            'The trust relationship between this workstation and the primary domain failed.';
    Win32ErrorCodes.ERROR_TRUST_FAILURE:
        Win32ErrorCodeDescription := 'The network logon failed.';
    Win32ErrorCodes.RPC_S_CALL_IN_PROGRESS:
        Win32ErrorCodeDescription :=
            'A remote procedure call is already in progress for this thread.';
    Win32ErrorCodes.ERROR_NETLOGON_NOT_STARTED:
        Win32ErrorCodeDescription :=
            'An attempt was made to logon, but the network logon service was not started.';
    Win32ErrorCodes.ERROR_ACCOUNT_EXPIRED:
        Win32ErrorCodeDescription := 'The users account has expired.';
    Win32ErrorCodes.ERROR_REDIRECTOR_HAS_OPEN_HANDLES:
        Win32ErrorCodeDescription := 'The redirector is in use and cannot be unloaded.';
    Win32ErrorCodes.ERROR_PRINTER_DRIVER_ALREADY_INSTALLED:
        Win32ErrorCodeDescription := 'The specified printer driver is already installed.';
    Win32ErrorCodes.ERROR_UNKNOWN_PORT:
        Win32ErrorCodeDescription := 'The specified port is unknown.';
    Win32ErrorCodes.ERROR_UNKNOWN_PRINTER_DRIVER:
        Win32ErrorCodeDescription := 'The printer driver is unknown.';
    Win32ErrorCodes.ERROR_UNKNOWN_PRINTPROCESSOR:
        Win32ErrorCodeDescription := 'The print processor is unknown.';
    Win32ErrorCodes.ERROR_INVALID_SEPARATOR_FILE:
        Win32ErrorCodeDescription := 'The specified separator file is invalid.';
    Win32ErrorCodes.ERROR_INVALID_PRIORITY:
        Win32ErrorCodeDescription := 'The specified priority is invalid.';
    Win32ErrorCodes.ERROR_INVALID_PRINTER_NAME:
        Win32ErrorCodeDescription := 'The printer name is invalid.';
    Win32ErrorCodes.ERROR_PRINTER_ALREADY_EXISTS:
        Win32ErrorCodeDescription := 'The printer already exists.';
    Win32ErrorCodes.ERROR_INVALID_PRINTER_COMMAND:
        Win32ErrorCodeDescription := 'The printer command is invalid.';
    Win32ErrorCodes.ERROR_INVALID_DATATYPE:
        Win32ErrorCodeDescription := 'The specified datatype is invalid.';
    Win32ErrorCodes.ERROR_INVALID_ENVIRONMENT:
        Win32ErrorCodeDescription := 'The environment specified is invalid.';
    Win32ErrorCodes.RPC_S_NO_MORE_BINDINGS:
        Win32ErrorCodeDescription := 'There are no more bindings.';
    Win32ErrorCodes.ERROR_NOLOGON_INTERDOMAIN_TRUST_ACCOUNT:
        Win32ErrorCodeDescription := 'The account used is an interdomain trust account. Use your global user account or local user account to access this server.';
    Win32ErrorCodes.ERROR_NOLOGON_WORKSTATION_TRUST_ACCOUNT:
        Win32ErrorCodeDescription := 'The account used is a computer account. Use your global user account or local user account to access this server.';
    Win32ErrorCodes.ERROR_NOLOGON_SERVER_TRUST_ACCOUNT:
        Win32ErrorCodeDescription := 'The account used is a server trust account. Use your global user account or local user account to access this server.';
    Win32ErrorCodes.ERROR_DOMAIN_TRUST_INCONSISTENT:
        Win32ErrorCodeDescription := 'The name or security ID (SID) of the domain specified is inconsistent with the trust information for that domain.';
    Win32ErrorCodes.ERROR_SERVER_HAS_OPEN_HANDLES:
        Win32ErrorCodeDescription := 'The server is in use and cannot be unloaded.';
    Win32ErrorCodes.ERROR_RESOURCE_DATA_NOT_FOUND:
        Win32ErrorCodeDescription :=
            'The specified image file did not contain a resource section.';
    Win32ErrorCodes.ERROR_RESOURCE_TYPE_NOT_FOUND:
        Win32ErrorCodeDescription :=
            'The specified resource type cannot be found in the image file.';
    Win32ErrorCodes.ERROR_RESOURCE_NAME_NOT_FOUND:
        Win32ErrorCodeDescription :=
            'The specified resource name cannot be found in the image file.';
    Win32ErrorCodes.ERROR_RESOURCE_LANG_NOT_FOUND:
        Win32ErrorCodeDescription :=
            'The specified resource language ID cannot be found in the image file.';
    Win32ErrorCodes.ERROR_NOT_ENOUGH_QUOTA:
        Win32ErrorCodeDescription := 'Not enough quota is available to process this command.';
    Win32ErrorCodes.RPC_S_NO_INTERFACES:
        Win32ErrorCodeDescription := 'No interfaces have been registered.';
    Win32ErrorCodes.RPC_S_CALL_CANCELLED:
        Win32ErrorCodeDescription := 'The remote procedure call was cancelled.';
    Win32ErrorCodes.RPC_S_BINDING_INCOMPLETE:
        Win32ErrorCodeDescription :=
            'The binding handle does not contain all required information.';
    Win32ErrorCodes.RPC_S_COMM_FAILURE:
        Win32ErrorCodeDescription :=
            'A communications failure occurred during a remote procedure call.';
    Win32ErrorCodes.RPC_S_UNSUPPORTED_AUTHN_LEVEL:
        Win32ErrorCodeDescription := 'The requested authentication level is not supported.';
    Win32ErrorCodes.RPC_S_NO_PRINC_NAME:
        Win32ErrorCodeDescription := 'No principal name registered.';
    Win32ErrorCodes.RPC_S_NOT_RPC_ERROR:
        Win32ErrorCodeDescription := 'The error specified is not a valid Windows RPC error code.';
    Win32ErrorCodes.RPC_S_UUID_LOCAL_ONLY:
        Win32ErrorCodeDescription :=
            'A UUID that is valid only on this computer has been allocated.';
    Win32ErrorCodes.RPC_S_SEC_PKG_ERROR:
        Win32ErrorCodeDescription := 'A security package specific error occurred.';
    Win32ErrorCodes.RPC_S_NOT_CANCELLED:
        Win32ErrorCodeDescription := 'Thread is not canceled.';
    Win32ErrorCodes.RPC_X_INVALID_ES_ACTION:
        Win32ErrorCodeDescription := 'Invalid operation on the encoding/decoding handle.';
    Win32ErrorCodes.RPC_X_WRONG_ES_VERSION:
        Win32ErrorCodeDescription := 'Incompatible version of the serializing package.';
    Win32ErrorCodes.RPC_X_WRONG_STUB_VERSION:
        Win32ErrorCodeDescription := 'Incompatible version of the RPC stub.';
    Win32ErrorCodes.RPC_X_INVALID_PIPE_OBJECT:
        Win32ErrorCodeDescription := 'The RPC pipe object is invalid or corrupted.';
    Win32ErrorCodes.RPC_X_WRONG_PIPE_ORDER:
        Win32ErrorCodeDescription := 'An invalid operation was attempted on an RPC pipe object.';
    Win32ErrorCodes.RPC_X_WRONG_PIPE_VERSION:
        Win32ErrorCodeDescription := 'Unsupported RPC pipe version.';
    Win32ErrorCodes.RPC_S_GROUP_MEMBER_NOT_FOUND:
        Win32ErrorCodeDescription := 'The group member was not found.';
    Win32ErrorCodes.EPT_S_CANT_CREATE:
        Win32ErrorCodeDescription := 'The endpoint mapper database entry could not be created.';
    Win32ErrorCodes.RPC_S_INVALID_OBJECT:
        Win32ErrorCodeDescription :=
            'The object universal unique identifier (UUID) is the nil UUID.';
    Win32ErrorCodes.ERROR_INVALID_TIME:
        Win32ErrorCodeDescription := 'The specified time is invalid.';
    Win32ErrorCodes.ERROR_INVALID_FORM_NAME:
        Win32ErrorCodeDescription := 'The specified form name is invalid.';
    Win32ErrorCodes.ERROR_INVALID_FORM_SIZE:
        Win32ErrorCodeDescription := 'The specified form size is invalid.';
    Win32ErrorCodes.ERROR_ALREADY_WAITING:
        Win32ErrorCodeDescription := 'The specified printer handle is already being waited on';
    Win32ErrorCodes.ERROR_PRINTER_DELETED:
        Win32ErrorCodeDescription := 'The specified printer has been deleted.';
    Win32ErrorCodes.ERROR_INVALID_PRINTER_STATE:
        Win32ErrorCodeDescription := 'The state of the printer is invalid.';
    Win32ErrorCodes.ERROR_PASSWORD_MUST_CHANGE:
        Win32ErrorCodeDescription :=
            'The users password must be changed before logging on the first time.';
    Win32ErrorCodes.ERROR_DOMAIN_CONTROLLER_NOT_FOUND:
        Win32ErrorCodeDescription := 'Could not find the domain controller for this domain.';
    Win32ErrorCodes.ERROR_ACCOUNT_LOCKED_OUT:
        Win32ErrorCodeDescription :=
            'The referenced account is currently locked out and may not be logged on to.';
    Win32ErrorCodes.OR_INVALID_OXID:
        Win32ErrorCodeDescription := 'The object exporter specified was not found.';
    Win32ErrorCodes.OR_INVALID_OID:
        Win32ErrorCodeDescription := 'The object specified was not found.';
    Win32ErrorCodes.OR_INVALID_SET:
        Win32ErrorCodeDescription := 'The object resolver set specified was not found.';
    Win32ErrorCodes.RPC_S_SEND_INCOMPLETE:
        Win32ErrorCodeDescription := 'Some data remains to be sent in the request buffer.';
    Win32ErrorCodes.RPC_S_INVALID_ASYNC_HANDLE:
        Win32ErrorCodeDescription := 'Invalid asynchronous remote procedure call handle.';
    Win32ErrorCodes.RPC_S_INVALID_ASYNC_CALL:
        Win32ErrorCodeDescription := 'Invalid asynchronous RPC call handle for this operation.';
    Win32ErrorCodes.RPC_X_PIPE_CLOSED:
        Win32ErrorCodeDescription := 'The RPC pipe object has already been closed.';
    Win32ErrorCodes.RPC_X_PIPE_DISCIPLINE_ERROR:
        Win32ErrorCodeDescription := 'The RPC call completed before all pipes were processed.';
    Win32ErrorCodes.RPC_X_PIPE_EMPTY:
        Win32ErrorCodeDescription := 'No more data is available from the RPC pipe.';
    Win32ErrorCodes.ERROR_NO_SITENAME:
        Win32ErrorCodeDescription := 'No site name is available for this machine.';
    Win32ErrorCodes.ERROR_CANT_ACCESS_FILE:
        Win32ErrorCodeDescription := 'The file can not be accessed by the system.';
    Win32ErrorCodes.ERROR_CANT_RESOLVE_FILENAME:
        Win32ErrorCodeDescription := 'The name of the file cannot be resolved by the system.';
    Win32ErrorCodes.RPC_S_ENTRY_TYPE_MISMATCH:
        Win32ErrorCodeDescription := 'The entry is not of the expected type.';
    Win32ErrorCodes.RPC_S_NOT_ALL_OBJS_EXPORTED:
        Win32ErrorCodeDescription :=
            'Not all object UUIDs could be exported to the specified entry.';
    Win32ErrorCodes.RPC_S_INTERFACE_NOT_EXPORTED:
        Win32ErrorCodeDescription := 'Interface could not be exported to the specified entry.';
    Win32ErrorCodes.RPC_S_PROFILE_NOT_ADDED:
        Win32ErrorCodeDescription := 'The specified profile entry could not be added.';
    Win32ErrorCodes.RPC_S_PRF_ELT_NOT_ADDED:
        Win32ErrorCodeDescription := 'The specified profile element could not be added.';
    Win32ErrorCodes.RPC_S_PRF_ELT_NOT_REMOVED:
        Win32ErrorCodeDescription := 'The specified profile element could not be removed.';
    Win32ErrorCodes.RPC_S_GRP_ELT_NOT_ADDED:
        Win32ErrorCodeDescription := 'The group element could not be added.';
    Win32ErrorCodes.RPC_S_GRP_ELT_NOT_REMOVED:
        Win32ErrorCodeDescription := 'The group element could not be removed.';
    Win32ErrorCodes.ERROR_KM_DRIVER_BLOCKED:
        Win32ErrorCodeDescription := 'The printer driver is not compatible with a policy enabled on your computer that blocks NT 4.0 drivers.';
    Win32ErrorCodes.ERROR_INVALID_PIXEL_FORMAT:
        Win32ErrorCodeDescription := 'The pixel format is invalid.';
    Win32ErrorCodes.ERROR_BAD_DRIVER:
        Win32ErrorCodeDescription := 'The specified driver is invalid.';
    Win32ErrorCodes.ERROR_INVALID_WINDOW_STYLE:
        Win32ErrorCodeDescription :=
            'The window style or class attribute is invalid for this operation.';
    Win32ErrorCodes.ERROR_METAFILE_NOT_SUPPORTED:
        Win32ErrorCodeDescription := 'The requested metafile operation is not supported.';
    Win32ErrorCodes.ERROR_TRANSFORM_NOT_SUPPORTED:
        Win32ErrorCodeDescription := 'The requested transformation operation is not supported.';
    Win32ErrorCodes.ERROR_CLIPPING_NOT_SUPPORTED:
        Win32ErrorCodeDescription := 'The requested clipping operation is not supported.';
    Win32ErrorCodes.ERROR_INVALID_CMM:
        Win32ErrorCodeDescription := 'The specified color management module is invalid.';
    Win32ErrorCodes.ERROR_INVALID_PROFILE:
        Win32ErrorCodeDescription := 'The specified color profile is invalid.';
    Win32ErrorCodes.ERROR_TAG_NOT_FOUND:
        Win32ErrorCodeDescription := 'The specified tag was not found.';
    Win32ErrorCodes.ERROR_TAG_NOT_PRESENT:
        Win32ErrorCodeDescription := 'A required tag is not present.';
    Win32ErrorCodes.ERROR_DUPLICATE_TAG:
        Win32ErrorCodeDescription := 'The specified tag is already present.';
    Win32ErrorCodes.ERROR_PROFILE_NOT_ASSOCIATED_WITH_DEVICE:
        Win32ErrorCodeDescription :=
            'The specified color profile is not associated with any device.';
    Win32ErrorCodes.ERROR_PROFILE_NOT_FOUND:
        Win32ErrorCodeDescription := 'The specified color profile was not found.';
    Win32ErrorCodes.ERROR_INVALID_COLORSPACE:
        Win32ErrorCodeDescription := 'The specified color space is invalid.';
    Win32ErrorCodes.ERROR_ICM_NOT_ENABLED:
        Win32ErrorCodeDescription := 'Image Color Management is not enabled.';
    Win32ErrorCodes.ERROR_DELETING_ICM_XFORM:
        Win32ErrorCodeDescription := 'There was an error while deleting the color transform.';
    Win32ErrorCodes.ERROR_INVALID_TRANSFORM:
        Win32ErrorCodeDescription := 'The specified color transform is invalid.';
    Win32ErrorCodes.ERROR_COLORSPACE_MISMATCH:
        Win32ErrorCodeDescription :=
            'The specified transform does not match the bitmaps color space.';
    Win32ErrorCodes.ERROR_INVALID_COLORINDEX:
        Win32ErrorCodeDescription :=
            'The specified named color index is not present in the profile.';
    Win32ErrorCodes.ERROR_CONNECTED_OTHER_PASSWORD:
        Win32ErrorCodeDescription := 'The network connection was made successfully, but the user had to be prompted for a password other than the one originally specified.';
    Win32ErrorCodes.ERROR_BAD_USERNAME:
        Win32ErrorCodeDescription := 'The specified username is invalid.';
    Win32ErrorCodes.ERROR_NOT_CONNECTED:
        Win32ErrorCodeDescription := 'This network connection does not exist.';
    Win32ErrorCodes.ERROR_OPEN_FILES:
        Win32ErrorCodeDescription := 'This network connection has files open or requests pending.';
    Win32ErrorCodes.ERROR_ACTIVE_CONNECTIONS:
        Win32ErrorCodeDescription := 'Active connections still exist.';
    Win32ErrorCodes.ERROR_DEVICE_IN_USE:
        Win32ErrorCodeDescription :=
            'The device is in use by an active process and cannot be disconnected.';
    Win32ErrorCodes.ERROR_PKINIT_FAILURE:
        Win32ErrorCodeDescription := 'The kerberos protocol encountered an error while validating the KDC certificate during smartcard logon.';
    Win32ErrorCodes.ERROR_SMARTCARD_SUBSYSTEM_FAILURE:
        Win32ErrorCodeDescription := 'The kerberos protocol encountered an error while attempting to utilize the smartcard subsystem.';
    Win32ErrorCodes.ERROR_UNKNOWN_PRINT_MONITOR:
        Win32ErrorCodeDescription := 'The specified print monitor is unknown.';
    Win32ErrorCodes.ERROR_PRINTER_DRIVER_IN_USE:
        Win32ErrorCodeDescription := 'The specified printer driver is currently in use.';
    Win32ErrorCodes.ERROR_SPOOL_FILE_NOT_FOUND:
        Win32ErrorCodeDescription := 'The spool file was not found.';
    Win32ErrorCodes.ERROR_SPL_NO_STARTDOC:
        Win32ErrorCodeDescription := 'A StartDocPrinter call was not issued.';
    Win32ErrorCodes.ERROR_SPL_NO_ADDJOB:
        Win32ErrorCodeDescription := 'An AddJob call was not issued.';
    Win32ErrorCodes.ERROR_PRINT_PROCESSOR_ALREADY_INSTALLED:
        Win32ErrorCodeDescription := 'The specified print processor has already been installed.';
    Win32ErrorCodes.ERROR_PRINT_MONITOR_ALREADY_INSTALLED:
        Win32ErrorCodeDescription := 'The specified print monitor has already been installed.';
    Win32ErrorCodes.ERROR_INVALID_PRINT_MONITOR:
        Win32ErrorCodeDescription :=
            'The specified print monitor does not have the required functions.';
    Win32ErrorCodes.ERROR_PRINT_MONITOR_IN_USE:
        Win32ErrorCodeDescription := 'The specified print monitor is currently in use.';
    Win32ErrorCodes.ERROR_PRINTER_HAS_JOBS_QUEUED:
        Win32ErrorCodeDescription :=
            'The requested operation is not allowed when there are jobs queued to the printer.';
    Win32ErrorCodes.ERROR_SUCCESS_REBOOT_REQUIRED:
        Win32ErrorCodeDescription := 'The requested operation is successful. Changes will not be effective until the system is rebooted.';
    Win32ErrorCodes.ERROR_SUCCESS_RESTART_REQUIRED:
        Win32ErrorCodeDescription := 'The requested operation is successful. Changes will not be effective until the service is restarted.';
    Win32ErrorCodes.ERROR_PRINTER_NOT_FOUND:
        Win32ErrorCodeDescription := 'No printers were found.';
    Win32ErrorCodes.ERROR_WINS_INTERNAL:
        Win32ErrorCodeDescription := 'WINS encountered an error while processing the command.';
    Win32ErrorCodes.ERROR_CAN_NOT_DEL_LOCAL_WINS:
        Win32ErrorCodeDescription := 'The local WINS can not be deleted.';
    Win32ErrorCodes.ERROR_STATIC_INIT:
        Win32ErrorCodeDescription := 'The importation from the file failed.';
    Win32ErrorCodes.ERROR_INC_BACKUP:
        Win32ErrorCodeDescription := 'The backup failed. Was a full backup done before?';
    Win32ErrorCodes.ERROR_FULL_BACKUP:
        Win32ErrorCodeDescription :=
            'The backup failed. Check the directory to which you are backing the database.';
    Win32ErrorCodes.ERROR_REC_NON_EXISTENT:
        Win32ErrorCodeDescription := 'The name does not exist in the WINS database.';
    Win32ErrorCodes.ERROR_RPL_NOT_ALLOWED:
        Win32ErrorCodeDescription := 'Replication with a nonconfigured partner is not allowed.';
    Win32ErrorCodes.ERROR_DHCP_ADDRESS_CONFLICT:
        Win32ErrorCodeDescription := 'The DHCP client has obtained an IP address that is already in use on the network. The local interface will be disabled until the DHCP client can obtain a new address.';
    Win32ErrorCodes.ERROR_WMI_GUID_NOT_FOUND:
        Win32ErrorCodeDescription :=
            'The GUID passed was not recognized as valid by a WMI data provider.';
    Win32ErrorCodes.ERROR_WMI_INSTANCE_NOT_FOUND:
        Win32ErrorCodeDescription :=
            'The instance name passed was not recognized as valid by a WMI data provider.';
    Win32ErrorCodes.ERROR_WMI_ITEMID_NOT_FOUND:
        Win32ErrorCodeDescription :=
            'The data item ID passed was not recognized as valid by a WMI data provider.';
    Win32ErrorCodes.ERROR_WMI_TRY_AGAIN:
        Win32ErrorCodeDescription :=
            'The WMI request could not be completed and should be retried.';
    Win32ErrorCodes.ERROR_WMI_DP_NOT_FOUND:
        Win32ErrorCodeDescription := 'The WMI data provider could not be located.';
    Win32ErrorCodes.ERROR_WMI_UNRESOLVED_INSTANCE_REF:
        Win32ErrorCodeDescription :=
            'The WMI data provider references an instance set that has not been registered.';
    Win32ErrorCodes.ERROR_WMI_ALREADY_ENABLED:
        Win32ErrorCodeDescription :=
            'The WMI data block or event notification has already been enabled.';
    Win32ErrorCodes.ERROR_WMI_GUID_DISCONNECTED:
        Win32ErrorCodeDescription := 'The WMI data block is no longer available.';
    Win32ErrorCodes.ERROR_WMI_SERVER_UNAVAILABLE:
        Win32ErrorCodeDescription := 'The WMI data service is not available.';
    Win32ErrorCodes.ERROR_WMI_DP_FAILED:
        Win32ErrorCodeDescription := 'The WMI data provider failed to carry out the request.';
    Win32ErrorCodes.ERROR_WMI_INVALID_MOF:
        Win32ErrorCodeDescription := 'The WMI MOF information is not valid.';
    Win32ErrorCodes.ERROR_WMI_INVALID_REGINFO:
        Win32ErrorCodeDescription := 'The WMI registration information is not valid.';
    Win32ErrorCodes.ERROR_WMI_ALREADY_DISABLED:
        Win32ErrorCodeDescription :=
            'The WMI data block or event notification has already been disabled.';
    Win32ErrorCodes.ERROR_WMI_READ_ONLY:
        Win32ErrorCodeDescription := 'The WMI data item or data block is read only.';
    Win32ErrorCodes.ERROR_WMI_SET_FAILURE:
        Win32ErrorCodeDescription := 'The WMI data item or data block could not be changed.';
    Win32ErrorCodes.ERROR_INVALID_MEDIA:
        Win32ErrorCodeDescription := 'The media identifier does not represent a valid medium.';
    Win32ErrorCodes.ERROR_INVALID_LIBRARY:
        Win32ErrorCodeDescription := 'The library identifier does not represent a valid library.';
    Win32ErrorCodes.ERROR_INVALID_MEDIA_POOL:
        Win32ErrorCodeDescription :=
            'The media pool identifier does not represent a valid media pool.';
    Win32ErrorCodes.ERROR_DRIVE_MEDIA_MISMATCH:
        Win32ErrorCodeDescription :=
            'The drive and medium are not compatible or exist in different libraries.';
    Win32ErrorCodes.ERROR_MEDIA_OFFLINE:
        Win32ErrorCodeDescription := 'The medium currently exists in an offline library and must be online to perform this operation.';
    Win32ErrorCodes.ERROR_LIBRARY_OFFLINE:
        Win32ErrorCodeDescription := 'The operation cannot be performed on an offline library.';
    Win32ErrorCodes.ERROR_EMPTY:
        Win32ErrorCodeDescription := 'The library, drive, or media pool is empty.';
    Win32ErrorCodes.ERROR_NOT_EMPTY:
        Win32ErrorCodeDescription :=
            'The library, drive, or media pool must be empty to perform this operation.';
    Win32ErrorCodes.ERROR_MEDIA_UNAVAILABLE:
        Win32ErrorCodeDescription :=
            'No media is currently available in this media pool or library.';
    Win32ErrorCodes.ERROR_RESOURCE_DISABLED:
        Win32ErrorCodeDescription := 'A resource required for this operation is disabled.';
    Win32ErrorCodes.ERROR_INVALID_CLEANER:
        Win32ErrorCodeDescription := 'The media identifier does not represent a valid cleaner.';
    Win32ErrorCodes.ERROR_UNABLE_TO_CLEAN:
        Win32ErrorCodeDescription := 'The drive cannot be cleaned or does not support cleaning.';
    Win32ErrorCodes.ERROR_OBJECT_NOT_FOUND:
        Win32ErrorCodeDescription := 'The object identifier does not represent a valid object.';
    Win32ErrorCodes.ERROR_DATABASE_FAILURE:
        Win32ErrorCodeDescription := 'Unable to read from or write to the database.';
    Win32ErrorCodes.ERROR_DATABASE_FULL:
        Win32ErrorCodeDescription := 'The database is full.';
    Win32ErrorCodes.ERROR_MEDIA_INCOMPATIBLE:
        Win32ErrorCodeDescription := 'The medium is not compatible with the device or media pool.';
    Win32ErrorCodes.ERROR_RESOURCE_NOT_PRESENT:
        Win32ErrorCodeDescription := 'The resource required for this operation does not exist.';
    Win32ErrorCodes.ERROR_INVALID_OPERATION:
        Win32ErrorCodeDescription := 'The operation identifier is not valid.';
    Win32ErrorCodes.ERROR_MEDIA_NOT_AVAILABLE:
        Win32ErrorCodeDescription := 'The media is not mounted or ready for use.';
    Win32ErrorCodes.ERROR_DEVICE_NOT_AVAILABLE:
        Win32ErrorCodeDescription := 'The device is not ready for use.';
    Win32ErrorCodes.ERROR_REQUEST_REFUSED:
        Win32ErrorCodeDescription := 'The operator or administrator has refused the request.';
    Win32ErrorCodes.ERROR_INVALID_DRIVE_OBJECT:
        Win32ErrorCodeDescription := 'The drive identifier does not represent a valid drive.';
    Win32ErrorCodes.ERROR_LIBRARY_FULL:
        Win32ErrorCodeDescription := 'Library is full. No slot is available for use.';
    Win32ErrorCodes.ERROR_MEDIUM_NOT_ACCESSIBLE:
        Win32ErrorCodeDescription := 'The transport cannot access the medium.';
    Win32ErrorCodes.ERROR_UNABLE_TO_LOAD_MEDIUM:
        Win32ErrorCodeDescription := 'Unable to load the medium into the drive.';
    Win32ErrorCodes.ERROR_UNABLE_TO_INVENTORY_DRIVE:
        Win32ErrorCodeDescription := 'Unable to retrieve status about the drive.';
    Win32ErrorCodes.ERROR_UNABLE_TO_INVENTORY_SLOT:
        Win32ErrorCodeDescription := 'Unable to retrieve status about the slot.';
    Win32ErrorCodes.ERROR_UNABLE_TO_INVENTORY_TRANSPORT:
        Win32ErrorCodeDescription := 'Unable to retrieve status about the transport.';
    Win32ErrorCodes.ERROR_TRANSPORT_FULL:
        Win32ErrorCodeDescription := 'Cannot use the transport because it is already in use.';
    Win32ErrorCodes.ERROR_CONTROLLING_IEPORT:
        Win32ErrorCodeDescription := 'Unable to open or close the inject/eject port.';
    Win32ErrorCodes.ERROR_UNABLE_TO_EJECT_MOUNTED_MEDIA:
        Win32ErrorCodeDescription := 'Unable to eject the media because it is in a drive.';
    Win32ErrorCodes.ERROR_CLEANER_SLOT_SET:
        Win32ErrorCodeDescription := 'A cleaner slot is already reserved.';
    Win32ErrorCodes.ERROR_CLEANER_SLOT_NOT_SET:
        Win32ErrorCodeDescription := 'A cleaner slot is not reserved.';
    Win32ErrorCodes.ERROR_CLEANER_CARTRIDGE_SPENT:
        Win32ErrorCodeDescription :=
            'The cleaner cartridge has performed the maximum number of drive cleanings.';
    Win32ErrorCodes.ERROR_UNEXPECTED_OMID:
        Win32ErrorCodeDescription := 'Unexpected on-medium identifier.';
    Win32ErrorCodes.ERROR_CANT_DELETE_LAST_ITEM:
        Win32ErrorCodeDescription :=
            'The last remaining item in this group or resource cannot be deleted.';
    Win32ErrorCodes.ERROR_MESSAGE_EXCEEDS_MAX_SIZE:
        Win32ErrorCodeDescription :=
            'The message provided exceeds the maximum size allowed for this parameter.';
    Win32ErrorCodes.ERROR_VOLUME_CONTAINS_SYS_FILES:
        Win32ErrorCodeDescription := 'The volume contains system or paging files.';
    Win32ErrorCodes.ERROR_INDIGENOUS_TYPE:
        Win32ErrorCodeDescription := 'The media type cannot be removed from this library since at least one drive in the library reports it can support this media type.';
    Win32ErrorCodes.ERROR_NO_SUPPORTING_DRIVES:
        Win32ErrorCodeDescription := 'This offline media cannot be mounted on this system since no enabled drives are present which can be used.';
    Win32ErrorCodes.ERROR_CLEANER_CARTRIDGE_INSTALLED:
        Win32ErrorCodeDescription := 'A cleaner cartridge is present in the tape library.';
    Win32ErrorCodes.ERROR_FILE_OFFLINE:
        Win32ErrorCodeDescription := 'The remote storage service was not able to recall the file.';
    Win32ErrorCodes.ERROR_REMOTE_STORAGE_NOT_ACTIVE:
        Win32ErrorCodeDescription := 'The remote storage service is not operational at this time.';
    Win32ErrorCodes.ERROR_REMOTE_STORAGE_MEDIA_ERROR:
        Win32ErrorCodeDescription := 'The remote storage service encountered a media error.';
    Win32ErrorCodes.ERROR_NOT_A_REPARSE_POINT:
        Win32ErrorCodeDescription := 'The file or directory is not a reparse point.';
    Win32ErrorCodes.ERROR_REPARSE_ATTRIBUTE_CONFLICT:
        Win32ErrorCodeDescription := 'The reparse point attribute cannot be set because it conflicts with an existing attribute.';
    Win32ErrorCodes.ERROR_INVALID_REPARSE_DATA:
        Win32ErrorCodeDescription := 'The data present in the reparse point buffer is invalid.';
    Win32ErrorCodes.ERROR_REPARSE_TAG_INVALID:
        Win32ErrorCodeDescription := 'The tag present in the reparse point buffer is invalid.';
    Win32ErrorCodes.ERROR_REPARSE_TAG_MISMATCH:
        Win32ErrorCodeDescription := 'There is a mismatch between the tag specified in the request and the tag present in the reparse point.';
    Win32ErrorCodes.ERROR_VOLUME_NOT_SIS_ENABLED:
        Win32ErrorCodeDescription := 'Single Instance Storage is not available on this volume.';
    Win32ErrorCodes.ERROR_DEPENDENT_RESOURCE_EXISTS:
        Win32ErrorCodeDescription := 'The cluster resource cannot be moved to another group because other resources are dependent on it.';
    Win32ErrorCodes.ERROR_DEPENDENCY_NOT_FOUND:
        Win32ErrorCodeDescription := 'The cluster resource dependency cannot be found.';
    Win32ErrorCodes.ERROR_DEPENDENCY_ALREADY_EXISTS:
        Win32ErrorCodeDescription := 'The cluster resource cannot be made dependent on the specified resource because it is already dependent.';
    Win32ErrorCodes.ERROR_RESOURCE_NOT_ONLINE:
        Win32ErrorCodeDescription := 'The cluster resource is not online.';
    Win32ErrorCodes.ERROR_HOST_NODE_NOT_AVAILABLE:
        Win32ErrorCodeDescription := 'A cluster node is not available for this operation.';
    Win32ErrorCodes.ERROR_RESOURCE_NOT_AVAILABLE:
        Win32ErrorCodeDescription := 'The cluster resource is not available.';
    Win32ErrorCodes.ERROR_RESOURCE_NOT_FOUND:
        Win32ErrorCodeDescription := 'The cluster resource could not be found.';
    Win32ErrorCodes.ERROR_SHUTDOWN_CLUSTER:
        Win32ErrorCodeDescription := 'The cluster is being shut down.';
    Win32ErrorCodes.ERROR_CANT_EVICT_ACTIVE_NODE:
        Win32ErrorCodeDescription :=
            'A cluster node cannot be evicted from the cluster unless the node is down.';
    Win32ErrorCodes.ERROR_OBJECT_ALREADY_EXISTS:
        Win32ErrorCodeDescription := 'The object already exists.';
    Win32ErrorCodes.ERROR_OBJECT_IN_LIST:
        Win32ErrorCodeDescription := 'The object is already in the list.';
    Win32ErrorCodes.ERROR_GROUP_NOT_AVAILABLE:
        Win32ErrorCodeDescription := 'The cluster group is not available for any new requests.';
    Win32ErrorCodes.ERROR_GROUP_NOT_FOUND:
        Win32ErrorCodeDescription := 'The cluster group could not be found.';
    Win32ErrorCodes.ERROR_GROUP_NOT_ONLINE:
        Win32ErrorCodeDescription :=
            'The operation could not be completed because the cluster group is not online.';
    Win32ErrorCodes.ERROR_HOST_NODE_NOT_RESOURCE_OWNER:
        Win32ErrorCodeDescription := 'The cluster node is not the owner of the resource.';
    Win32ErrorCodes.ERROR_HOST_NODE_NOT_GROUP_OWNER:
        Win32ErrorCodeDescription := 'The cluster node is not the owner of the group.';
    Win32ErrorCodes.ERROR_RESMON_CREATE_FAILED:
        Win32ErrorCodeDescription :=
            'The cluster resource could not be created in the specified resource monitor.';
    Win32ErrorCodes.ERROR_RESMON_ONLINE_FAILED:
        Win32ErrorCodeDescription :=
            'The cluster resource could not be brought online by the resource monitor.';
    Win32ErrorCodes.ERROR_RESOURCE_ONLINE:
        Win32ErrorCodeDescription :=
            'The operation could not be completed because the cluster resource is online.';
    Win32ErrorCodes.ERROR_QUORUM_RESOURCE:
        Win32ErrorCodeDescription := 'The cluster resource could not be deleted or brought offline because it is the quorum resource.';
    Win32ErrorCodes.ERROR_NOT_QUORUM_CAPABLE:
        Win32ErrorCodeDescription := 'The cluster could not make the specified resource a quorum resource because it is not capable of being a quorum resource.';
    Win32ErrorCodes.ERROR_CLUSTER_SHUTTING_DOWN:
        Win32ErrorCodeDescription := 'The cluster software is shutting down.';
    Win32ErrorCodes.ERROR_INVALID_STATE:
        Win32ErrorCodeDescription :=
            'The group or resource is not in the correct state to perform the requested operation.';
    Win32ErrorCodes.ERROR_RESOURCE_PROPERTIES_STORED:
        Win32ErrorCodeDescription := 'The properties were stored but not all changes will take effect until the next time the resource is brought online.';
    Win32ErrorCodes.ERROR_NOT_QUORUM_CLASS:
        Win32ErrorCodeDescription := 'The cluster could not make the specified resource a quorum resource because it does not belong to a shared storage class.';
    Win32ErrorCodes.ERROR_CORE_RESOURCE:
        Win32ErrorCodeDescription :=
            'The cluster resource could not be deleted since it is a core resource.';
    Win32ErrorCodes.ERROR_QUORUM_RESOURCE_ONLINE_FAILED:
        Win32ErrorCodeDescription := 'The quorum resource failed to come online.';
    Win32ErrorCodes.ERROR_QUORUMLOG_OPEN_FAILED:
        Win32ErrorCodeDescription :=
            'The quorum log could not be created or mounted successfully.';
    Win32ErrorCodes.ERROR_CLUSTERLOG_CORRUPT:
        Win32ErrorCodeDescription := 'The cluster log is corrupt.';
    Win32ErrorCodes.ERROR_CLUSTERLOG_RECORD_EXCEEDS_MAXSIZE:
        Win32ErrorCodeDescription :=
            'The record could not be written to the cluster log since it exceeds the maximum size.';
    Win32ErrorCodes.ERROR_CLUSTERLOG_EXCEEDS_MAXSIZE:
        Win32ErrorCodeDescription := 'The cluster log exceeds its maximum size.';
    Win32ErrorCodes.ERROR_CLUSTERLOG_CHKPOINT_NOT_FOUND:
        Win32ErrorCodeDescription := 'No checkpoint record was found in the cluster log.';
    Win32ErrorCodes.ERROR_CLUSTERLOG_NOT_ENOUGH_SPACE:
        Win32ErrorCodeDescription :=
            'The minimum required disk space needed for logging is not available.';
    Win32ErrorCodes.ERROR_QUORUM_OWNER_ALIVE:
        Win32ErrorCodeDescription := 'The cluster node failed to take control of the quorum resource because the resource is owned by another active node.';
    Win32ErrorCodes.ERROR_NETWORK_NOT_AVAILABLE:
        Win32ErrorCodeDescription := 'A cluster network is not available for this operation.';
    Win32ErrorCodes.ERROR_NODE_NOT_AVAILABLE:
        Win32ErrorCodeDescription := 'A cluster node is not available for this operation.';
    Win32ErrorCodes.ERROR_ALL_NODES_NOT_AVAILABLE:
        Win32ErrorCodeDescription :=
            'All cluster nodes must be running to perform this operation.';
    Win32ErrorCodes.ERROR_RESOURCE_FAILED:
        Win32ErrorCodeDescription := 'A cluster resource failed.';
    Win32ErrorCodes.ERROR_CLUSTER_INVALID_NODE:
        Win32ErrorCodeDescription := 'The cluster node is not valid.';
    Win32ErrorCodes.ERROR_CLUSTER_NODE_EXISTS:
        Win32ErrorCodeDescription := 'The cluster node already exists.';
    Win32ErrorCodes.ERROR_CLUSTER_JOIN_IN_PROGRESS:
        Win32ErrorCodeDescription := 'A node is in the process of joining the cluster.';
    Win32ErrorCodes.ERROR_CLUSTER_NODE_NOT_FOUND:
        Win32ErrorCodeDescription := 'The cluster node was not found.';
    Win32ErrorCodes.ERROR_CLUSTER_LOCAL_NODE_NOT_FOUND:
        Win32ErrorCodeDescription := 'The cluster local node information was not found.';
    Win32ErrorCodes.ERROR_CLUSTER_NETWORK_EXISTS:
        Win32ErrorCodeDescription := 'The cluster network already exists.';
    Win32ErrorCodes.ERROR_CLUSTER_NETWORK_NOT_FOUND:
        Win32ErrorCodeDescription := 'The cluster network was not found.';
    Win32ErrorCodes.ERROR_CLUSTER_NETINTERFACE_EXISTS:
        Win32ErrorCodeDescription := 'The cluster network interface already exists.';
    Win32ErrorCodes.ERROR_CLUSTER_NETINTERFACE_NOT_FOUND:
        Win32ErrorCodeDescription := 'The cluster network interface was not found.';
    Win32ErrorCodes.ERROR_CLUSTER_INVALID_REQUEST:
        Win32ErrorCodeDescription := 'The cluster request is not valid for this object.';
    Win32ErrorCodes.ERROR_CLUSTER_INVALID_NETWORK_PROVIDER:
        Win32ErrorCodeDescription := 'The cluster network provider is not valid.';
    Win32ErrorCodes.ERROR_CLUSTER_NODE_DOWN:
        Win32ErrorCodeDescription := 'The cluster node is down.';
    Win32ErrorCodes.ERROR_CLUSTER_NODE_UNREACHABLE:
        Win32ErrorCodeDescription := 'The cluster node is not reachable.';
    Win32ErrorCodes.ERROR_CLUSTER_NODE_NOT_MEMBER:
        Win32ErrorCodeDescription := 'The cluster node is not a member of the cluster.';
    Win32ErrorCodes.ERROR_CLUSTER_JOIN_NOT_IN_PROGRESS:
        Win32ErrorCodeDescription := 'A cluster join operation is not in progress.';
    Win32ErrorCodes.ERROR_CLUSTER_INVALID_NETWORK:
        Win32ErrorCodeDescription := 'The cluster network is not valid.';
    Win32ErrorCodes.ERROR_CLUSTER_NODE_UP:
        Win32ErrorCodeDescription := 'The cluster node is up.';
    Win32ErrorCodes.ERROR_CLUSTER_IPADDR_IN_USE:
        Win32ErrorCodeDescription := 'The cluster IP address is already in use.';
    Win32ErrorCodes.ERROR_CLUSTER_NODE_NOT_PAUSED:
        Win32ErrorCodeDescription := 'The cluster node is not paused.';
    Win32ErrorCodes.ERROR_CLUSTER_NO_SECURITY_CONTEXT:
        Win32ErrorCodeDescription := 'No cluster security context is available.';
    Win32ErrorCodes.ERROR_CLUSTER_NETWORK_NOT_INTERNAL:
        Win32ErrorCodeDescription :=
            'The cluster network is not configured for internal cluster communication.';
    Win32ErrorCodes.ERROR_CLUSTER_NODE_ALREADY_UP:
        Win32ErrorCodeDescription := 'The cluster node is already up.';
    Win32ErrorCodes.ERROR_CLUSTER_NODE_ALREADY_DOWN:
        Win32ErrorCodeDescription := 'The cluster node is already down.';
    Win32ErrorCodes.ERROR_CLUSTER_NETWORK_ALREADY_ONLINE:
        Win32ErrorCodeDescription := 'The cluster network is already online.';
    Win32ErrorCodes.ERROR_CLUSTER_NETWORK_ALREADY_OFFLINE:
        Win32ErrorCodeDescription := 'The cluster network is already offline.';
    Win32ErrorCodes.ERROR_CLUSTER_NODE_ALREADY_MEMBER:
        Win32ErrorCodeDescription := 'The cluster node is already a member of the cluster.';
    Win32ErrorCodes.ERROR_CLUSTER_LAST_INTERNAL_NETWORK:
        Win32ErrorCodeDescription := 'The cluster network is the only one configured for internal cluster communication between two or more active cluster nodes. The internal communication capability cannot be removed from the network.';
    Win32ErrorCodes.ERROR_CLUSTER_NETWORK_HAS_DEPENDENTS:
        Win32ErrorCodeDescription := 'One or more cluster resources depend on the network to provide service to clients. The client access capability cannot be removed from the network.';
    Win32ErrorCodes.ERROR_INVALID_OPERATION_ON_QUORUM:
        Win32ErrorCodeDescription := 'This operation cannot be performed on the cluster resource as it the quorum resource. You may not bring the quorum resource offline or modify its possible owners list.';
    Win32ErrorCodes.ERROR_DEPENDENCY_NOT_ALLOWED:
        Win32ErrorCodeDescription :=
            'The cluster quorum resource is not allowed to have any dependencies.';
    Win32ErrorCodes.ERROR_CLUSTER_NODE_PAUSED:
        Win32ErrorCodeDescription := 'The cluster node is paused.';
    Win32ErrorCodes.ERROR_NODE_CANT_HOST_RESOURCE:
        Win32ErrorCodeDescription :=
            'The cluster resource cannot be brought online. The owner node cannot run this resource.';
    Win32ErrorCodes.ERROR_CLUSTER_NODE_NOT_READY:
        Win32ErrorCodeDescription :=
            'The cluster node is not ready to perform the requested operation.';
    Win32ErrorCodes.ERROR_CLUSTER_NODE_SHUTTING_DOWN:
        Win32ErrorCodeDescription := 'The cluster node is shutting down.';
    Win32ErrorCodes.ERROR_CLUSTER_JOIN_ABORTED:
        Win32ErrorCodeDescription := 'The cluster join operation was aborted.';
    Win32ErrorCodes.ERROR_CLUSTER_INCOMPATIBLE_VERSIONS:
        Win32ErrorCodeDescription := 'The cluster join operation failed due to incompatible software versions between the joining node and its sponsor.';
    Win32ErrorCodes.ERROR_CLUSTER_MAXNUM_OF_RESOURCES_EXCEEDED:
        Win32ErrorCodeDescription := 'This resource cannot be created because the cluster has reached the limit on the number of resources it can monitor.';
    Win32ErrorCodes.ERROR_CLUSTER_SYSTEM_CONFIG_CHANGED:
        Win32ErrorCodeDescription := 'The system configuration changed during the cluster join or form operation. The join or form operation was aborted.';
    Win32ErrorCodes.ERROR_CLUSTER_RESOURCE_TYPE_NOT_FOUND:
        Win32ErrorCodeDescription := 'The specified resource type was not found.';
    Win32ErrorCodes.ERROR_CLUSTER_RESTYPE_NOT_SUPPORTED:
        Win32ErrorCodeDescription := 'The specified node does not support a resource of this type. This may be due to version inconsistencies or due to the absence of the resource DLL on this node.';
    Win32ErrorCodes.ERROR_CLUSTER_RESNAME_NOT_FOUND:
        Win32ErrorCodeDescription := 'The specified resource name is supported by this resource DLL. This may be due to a bad (or changed) name supplied to the resource DLL.';
    Win32ErrorCodes.ERROR_CLUSTER_NO_RPC_PACKAGES_REGISTERED:
        Win32ErrorCodeDescription :=
            'No authentication package could be registered with the RPC server.';
    Win32ErrorCodes.ERROR_CLUSTER_OWNER_NOT_IN_PREFLIST:
        Win32ErrorCodeDescription := 'You cannot bring the group online because the owner of the group is not in the preferred list for the group. To change the owner node for the group, move the group.';
    Win32ErrorCodes.ERROR_CLUSTER_DATABASE_SEQMISMATCH:
        Win32ErrorCodeDescription := 'The join operation failed because the cluster database sequence number has changed or is incompatible with the locker node. This may happen during a join operation if the cluster database was changing during the join.';
    Win32ErrorCodes.ERROR_RESMON_INVALID_STATE:
        Win32ErrorCodeDescription := 'The resource monitor will not allow the fail operation to be performed while the resource is in its current state. This may happen if the resource is in a pending state.';
    Win32ErrorCodes.ERROR_CLUSTER_GUM_NOT_LOCKER:
        Win32ErrorCodeDescription :=
            'A non locker code got a request to reserve the lock for making global updates.';
    Win32ErrorCodes.ERROR_QUORUM_DISK_NOT_FOUND:
        Win32ErrorCodeDescription :=
            'The quorum disk could not be located by the cluster service.';
    Win32ErrorCodes.ERROR_DATABASE_BACKUP_CORRUPT:
        Win32ErrorCodeDescription := 'The backup up cluster database is possibly corrupt.';
    Win32ErrorCodes.ERROR_CLUSTER_NODE_ALREADY_HAS_DFS_ROOT:
        Win32ErrorCodeDescription := 'A DFS root already exists in this cluster node.';
    Win32ErrorCodes.ERROR_RESOURCE_PROPERTY_UNCHANGEABLE:
        Win32ErrorCodeDescription := 'An attempt to modify a resource property failed because it conflicts with another existing property.';
    Win32ErrorCodes.ERROR_CLUSTER_MEMBERSHIP_INVALID_STATE:
        Win32ErrorCodeDescription := 'An operation was attempted that is incompatible with the current membership state of the node.';
    Win32ErrorCodes.ERROR_CLUSTER_QUORUMLOG_NOT_FOUND:
        Win32ErrorCodeDescription := 'The quorum resource does not contain the quorum log.';
    Win32ErrorCodes.ERROR_CLUSTER_MEMBERSHIP_HALT:
        Win32ErrorCodeDescription :=
            'The membership engine requested shutdown of the cluster service on this node.';
    Win32ErrorCodes.ERROR_CLUSTER_INSTANCE_ID_MISMATCH:
        Win32ErrorCodeDescription := 'The join operation failed because the cluster instance ID of the joining node does not match the cluster instance ID of the sponsor node.';
    Win32ErrorCodes.ERROR_CLUSTER_NETWORK_NOT_FOUND_FOR_IP:
        Win32ErrorCodeDescription := 'A matching network for the specified IP address could not be found. Please also specify a subnet mask and a cluster network.';
    Win32ErrorCodes.ERROR_CLUSTER_PROPERTY_DATA_TYPE_MISMATCH:
        Win32ErrorCodeDescription := 'The actual data type of the property did not match the expected data type of the property.';
    Win32ErrorCodes.ERROR_CLUSTER_EVICT_WITHOUT_CLEANUP:
        Win32ErrorCodeDescription := 'The cluster node was evicted from the cluster successfully. The node was not cleaned up because it does not support the evict cleanup functionality.';
    Win32ErrorCodes.ERROR_ENCRYPTION_FAILED:
        Win32ErrorCodeDescription := 'The specified file could not be encrypted.';
    Win32ErrorCodes.ERROR_DECRYPTION_FAILED:
        Win32ErrorCodeDescription := 'The specified file could not be decrypted.';
    Win32ErrorCodes.ERROR_FILE_ENCRYPTED:
        Win32ErrorCodeDescription :=
            'The specified file is encrypted and the user does not have the ability to decrypt it.';
    Win32ErrorCodes.ERROR_NO_RECOVERY_POLICY:
        Win32ErrorCodeDescription :=
            'There is no valid encryption recovery policy configured for this system.';
    Win32ErrorCodes.ERROR_NO_EFS:
        Win32ErrorCodeDescription :=
            'The required encryption driver is not loaded for this system.';
    Win32ErrorCodes.ERROR_WRONG_EFS:
        Win32ErrorCodeDescription :=
            'The file was encrypted with a different encryption driver than is currently loaded.';
    Win32ErrorCodes.ERROR_NO_USER_KEYS:
        Win32ErrorCodeDescription := 'There are no EFS keys defined for the user.';
    Win32ErrorCodes.ERROR_FILE_NOT_ENCRYPTED:
        Win32ErrorCodeDescription := 'The specified file is not encrypted.';
    Win32ErrorCodes.ERROR_NOT_EXPORT_FORMAT:
        Win32ErrorCodeDescription := 'The specified file is not in the defined EFS export format.';
    Win32ErrorCodes.ERROR_FILE_READ_ONLY:
        Win32ErrorCodeDescription := 'The specified file is read only.';
    Win32ErrorCodes.ERROR_DIR_EFS_DISALLOWED:
        Win32ErrorCodeDescription := 'The directory has been disabled for encryption.';
    Win32ErrorCodes.ERROR_EFS_SERVER_NOT_TRUSTED:
        Win32ErrorCodeDescription := 'The server is not trusted for remote encryption operation.';
    Win32ErrorCodes.ERROR_BAD_RECOVERY_POLICY:
        Win32ErrorCodeDescription :=
            'Recovery policy configured for this system contains invalid recovery certificate.';
    Win32ErrorCodes.ERROR_EFS_ALG_BLOB_TOO_BIG:
        Win32ErrorCodeDescription := 'The encryption algorithm used on the source file needs a bigger key buffer than the one on the destination file.';
    Win32ErrorCodes.ERROR_VOLUME_NOT_SUPPORT_EFS:
        Win32ErrorCodeDescription := 'The disk partition does not support file encryption.';
    Win32ErrorCodes.ERROR_NO_BROWSER_SERVERS_FOUND:
        Win32ErrorCodeDescription :=
            'The list of servers for this workgroup is not currently available.';
    Win32ErrorCodes.SCHED_E_SERVICE_NOT_LOCALSYSTEM:
        Win32ErrorCodeDescription := 'The Task Scheduler service must be configured to run in the System account to function properly. Individual tasks may be configured to run in other accounts.';
    Win32ErrorCodes.ERROR_CTX_WINSTATION_NAME_INVALID:
        Win32ErrorCodeDescription := 'The specified session name is invalid.';
    Win32ErrorCodes.ERROR_CTX_INVALID_PD:
        Win32ErrorCodeDescription := 'The specified protocol driver is invalid.';
    Win32ErrorCodes.ERROR_CTX_PD_NOT_FOUND:
        Win32ErrorCodeDescription :=
            'The specified protocol driver was not found in the system path.';
    Win32ErrorCodes.ERROR_CTX_WD_NOT_FOUND:
        Win32ErrorCodeDescription :=
            'The specified terminal connection driver was not found in the system path.';
    Win32ErrorCodes.ERROR_CTX_CANNOT_MAKE_EVENTLOG_ENTRY:
        Win32ErrorCodeDescription :=
            'A registry key for event logging could not be created for this session.';
    Win32ErrorCodes.ERROR_CTX_SERVICE_NAME_COLLISION:
        Win32ErrorCodeDescription := 'A service with the same name already exists on the system.';
    Win32ErrorCodes.ERROR_CTX_CLOSE_PENDING:
        Win32ErrorCodeDescription := 'A close operation is pending on the session.';
    Win32ErrorCodes.ERROR_CTX_NO_OUTBUF:
        Win32ErrorCodeDescription := 'There are no free output buffers available.';
    Win32ErrorCodes.ERROR_CTX_MODEM_INF_NOT_FOUND:
        Win32ErrorCodeDescription := 'The MODEM.INF file was not found.';
    Win32ErrorCodes.ERROR_CTX_INVALID_MODEMNAME:
        Win32ErrorCodeDescription := 'The modem name was not found in MODEM.INF.';
    Win32ErrorCodes.ERROR_CTX_MODEM_RESPONSE_ERROR:
        Win32ErrorCodeDescription := 'The modem did not accept the command sent to it. Verify that the configured modem name matches the attached modem.';
    Win32ErrorCodes.ERROR_CTX_MODEM_RESPONSE_TIMEOUT:
        Win32ErrorCodeDescription := 'The modem did not respond to the command sent to it. Verify that the modem is properly cabled and powered on.';
    Win32ErrorCodes.ERROR_CTX_MODEM_RESPONSE_NO_CARRIER:
        Win32ErrorCodeDescription :=
            'Carrier detect has failed or carrier has been dropped due to disconnect.';
    Win32ErrorCodes.ERROR_CTX_MODEM_RESPONSE_NO_DIALTONE:
        Win32ErrorCodeDescription := 'Dial tone not detected within the required time. Verify that the phone cable is properly attached and functional.';
    Win32ErrorCodes.ERROR_CTX_MODEM_RESPONSE_BUSY:
        Win32ErrorCodeDescription := 'Busy signal detected at remote site on callback.';
    Win32ErrorCodes.ERROR_CTX_MODEM_RESPONSE_VOICE:
        Win32ErrorCodeDescription := 'Voice detected at remote site on callback.';
    Win32ErrorCodes.ERROR_CTX_TD_ERROR:
        Win32ErrorCodeDescription := 'Transport driver error';
    Win32ErrorCodes.ERROR_CTX_WINSTATION_NOT_FOUND:
        Win32ErrorCodeDescription := 'The specified session cannot be found.';
    Win32ErrorCodes.ERROR_CTX_WINSTATION_ALREADY_EXISTS:
        Win32ErrorCodeDescription := 'The specified session name is already in use.';
    Win32ErrorCodes.ERROR_CTX_WINSTATION_BUSY:
        Win32ErrorCodeDescription := 'The requested operation cannot be completed because the terminal connection is currently busy processing a connect, disconnect, reset, or delete operation.';
    Win32ErrorCodes.ERROR_CTX_BAD_VIDEO_MODE:
        Win32ErrorCodeDescription := 'An attempt has been made to connect to a session whose video mode is not supported by the current client.';
    Win32ErrorCodes.ERROR_CTX_GRAPHICS_INVALID:
        Win32ErrorCodeDescription := 'The application attempted to enable DOS graphics mode. DOS graphics mode is not supported.';
    Win32ErrorCodes.ERROR_CTX_LOGON_DISABLED:
        Win32ErrorCodeDescription :=
            'Your interactive logon privilege has been disabled. Please contact your administrator.';
    Win32ErrorCodes.ERROR_CTX_NOT_CONSOLE:
        Win32ErrorCodeDescription := 'The requested operation can be performed only on the system console. This is most often the result of a driver or system DLL requiring direct console access.';
    Win32ErrorCodes.ERROR_CTX_CLIENT_QUERY_TIMEOUT:
        Win32ErrorCodeDescription := 'The client failed to respond to the server connect message.';
    Win32ErrorCodes.ERROR_CTX_CONSOLE_DISCONNECT:
        Win32ErrorCodeDescription := 'Disconnecting the console session is not supported.';
    Win32ErrorCodes.ERROR_CTX_CONSOLE_CONNECT:
        Win32ErrorCodeDescription :=
            'Reconnecting a disconnected session to the console is not supported.';
    Win32ErrorCodes.ERROR_CTX_SHADOW_DENIED:
        Win32ErrorCodeDescription := 'The request to control another session remotely was denied.';
    Win32ErrorCodes.ERROR_CTX_WINSTATION_ACCESS_DENIED:
        Win32ErrorCodeDescription := 'The requested session access is denied.';
    Win32ErrorCodes.ERROR_CTX_INVALID_WD:
        Win32ErrorCodeDescription := 'The specified terminal connection driver is invalid.';
    Win32ErrorCodes.ERROR_CTX_SHADOW_INVALID:
        Win32ErrorCodeDescription := 'The requested session cannot be controlled remotely. This may be because the session is disconnected or does not currently have a user logged on.';
    Win32ErrorCodes.ERROR_CTX_SHADOW_DISABLED:
        Win32ErrorCodeDescription :=
            'The requested session is not configured to allow remote control.';
    Win32ErrorCodes.ERROR_CTX_CLIENT_LICENSE_IN_USE:
        Win32ErrorCodeDescription := 'Your request to connect to this Terminal Server has been rejected. Your Terminal Server client license number is currently being used by another user. Please call your system administrator to obtain a unique license number.';
    Win32ErrorCodes.ERROR_CTX_CLIENT_LICENSE_NOT_SET:
        Win32ErrorCodeDescription := 'Your request to connect to this Terminal Server has been rejected. Your Terminal Server client license number has not been entered for this copy of the Terminal Server client. Please contact your system administrator.';
    Win32ErrorCodes.ERROR_CTX_LICENSE_NOT_AVAILABLE:
        Win32ErrorCodeDescription :=
            'The system has reached its licensed logon limit. Please try again later.';
    Win32ErrorCodes.ERROR_CTX_LICENSE_CLIENT_INVALID:
        Win32ErrorCodeDescription := 'The client you are using is not licensed to use this system. Your logon request is denied.';
    Win32ErrorCodes.ERROR_CTX_LICENSE_EXPIRED:
        Win32ErrorCodeDescription :=
            'The system license has expired. Your logon request is denied.';
    Win32ErrorCodes.ERROR_CTX_SHADOW_NOT_RUNNING:
        Win32ErrorCodeDescription := 'Remote control could not be terminated because the specified session is not currently being remotely controlled.';
    Win32ErrorCodes.FRS_ERR_INVALID_API_SEQUENCE:
        Win32ErrorCodeDescription := 'The file replication service API was called incorrectly.';
    Win32ErrorCodes.FRS_ERR_STARTING_SERVICE:
        Win32ErrorCodeDescription := 'The file replication service cannot be started.';
    Win32ErrorCodes.FRS_ERR_STOPPING_SERVICE:
        Win32ErrorCodeDescription := 'The file replication service cannot be stopped.';
    Win32ErrorCodes.FRS_ERR_INTERNAL_API:
        Win32ErrorCodeDescription := 'The file replication service API terminated the request. The event log may have more information.';
    Win32ErrorCodes.FRS_ERR_INTERNAL:
        Win32ErrorCodeDescription := 'The file replication service terminated the request. The event log may have more information.';
    Win32ErrorCodes.FRS_ERR_SERVICE_COMM:
        Win32ErrorCodeDescription := 'The file replication service cannot be contacted. The event log may have more information.';
    Win32ErrorCodes.FRS_ERR_INSUFFICIENT_PRIV:
        Win32ErrorCodeDescription := 'The file replication service cannot satisfy the request because the user has insufficient privileges. The event log may have more information.';
    Win32ErrorCodes.FRS_ERR_AUTHENTICATION:
        Win32ErrorCodeDescription := 'The file replication service cannot satisfy the request because authenticated RPC is not available. The event log may have more information.';
    Win32ErrorCodes.FRS_ERR_PARENT_INSUFFICIENT_PRIV:
        Win32ErrorCodeDescription := 'The file replication service cannot satisfy the request because the user has insufficient privileges on the domain controller. The event log may have more information.';
    Win32ErrorCodes.FRS_ERR_PARENT_AUTHENTICATION:
        Win32ErrorCodeDescription := 'The file replication service cannot satisfy the request because authenticated RPC is not available on the domain controller. The event log may have more information.';
    Win32ErrorCodes.FRS_ERR_CHILD_TO_PARENT_COMM:
        Win32ErrorCodeDescription := 'The file replication service cannot communicate with the file replication service on the domain controller. The event log may have more information.';
    Win32ErrorCodes.FRS_ERR_PARENT_TO_CHILD_COMM:
        Win32ErrorCodeDescription := 'The file replication service on the domain controller cannot communicate with the file replication service on this computer. The event log may have more information.';
    Win32ErrorCodes.FRS_ERR_SYSVOL_POPULATE:
        Win32ErrorCodeDescription := 'The file replication service cannot populate the system volume because of an internal error. The event log may have more information.';
    Win32ErrorCodes.FRS_ERR_SYSVOL_POPULATE_TIMEOUT:
        Win32ErrorCodeDescription := 'The file replication service cannot populate the system volume because of an internal timeout. The event log may have more information.';
    Win32ErrorCodes.FRS_ERR_SYSVOL_IS_BUSY:
        Win32ErrorCodeDescription := 'The file replication service cannot process the request. The system volume is busy with a previous request.';
    Win32ErrorCodes.FRS_ERR_SYSVOL_DEMOTE:
        Win32ErrorCodeDescription := 'The file replication service cannot stop replicating the system volume because of an internal error. The event log may have more information.';
    Win32ErrorCodes.FRS_ERR_INVALID_SERVICE_PARAMETER:
        Win32ErrorCodeDescription := 'The file replication service detected an invalid parameter.';
    Win32ErrorCodes.ERROR_DS_NOT_INSTALLED:
        Win32ErrorCodeDescription := 'An error occurred while installing the directory service. For more information, see the event log.';
    Win32ErrorCodes.ERROR_DS_MEMBERSHIP_EVALUATED_LOCALLY:
        Win32ErrorCodeDescription := 'The directory service evaluated group memberships locally.';
    Win32ErrorCodes.ERROR_DS_NO_ATTRIBUTE_OR_VALUE:
        Win32ErrorCodeDescription :=
            'The specified directory service attribute or value does not exist.';
    Win32ErrorCodes.ERROR_DS_INVALID_ATTRIBUTE_SYNTAX:
        Win32ErrorCodeDescription :=
            'The attribute syntax specified to the directory service is invalid.';
    Win32ErrorCodes.ERROR_DS_ATTRIBUTE_TYPE_UNDEFINED:
        Win32ErrorCodeDescription :=
            'The attribute type specified to the directory service is not defined.';
    Win32ErrorCodes.ERROR_DS_ATTRIBUTE_OR_VALUE_EXISTS:
        Win32ErrorCodeDescription :=
            'The specified directory service attribute or value already exists.';
    Win32ErrorCodes.ERROR_DS_BUSY:
        Win32ErrorCodeDescription := 'The directory service is busy.';
    Win32ErrorCodes.ERROR_DS_UNAVAILABLE:
        Win32ErrorCodeDescription := 'The directory service is unavailable.';
    Win32ErrorCodes.ERROR_DS_NO_RIDS_ALLOCATED:
        Win32ErrorCodeDescription :=
            'The directory service was unable to allocate a relative identifier.';
    Win32ErrorCodes.ERROR_DS_NO_MORE_RIDS:
        Win32ErrorCodeDescription :=
            'The directory service has exhausted the pool of relative identifiers.';
    Win32ErrorCodes.ERROR_DS_INCORRECT_ROLE_OWNER:
        Win32ErrorCodeDescription := 'The requested operation could not be performed because the directory service is not the master for that type of operation.';
    Win32ErrorCodes.ERROR_DS_RIDMGR_INIT_ERROR:
        Win32ErrorCodeDescription := 'The directory service was unable to initialize the subsystem that allocates relative identifiers.';
    Win32ErrorCodes.ERROR_DS_OBJ_CLASS_VIOLATION:
        Win32ErrorCodeDescription := 'The requested operation did not satisfy one or more constraints associated with the class of the object.';
    Win32ErrorCodes.ERROR_DS_CANT_ON_NON_LEAF:
        Win32ErrorCodeDescription :=
            'The directory service can perform the requested operation only on a leaf object.';
    Win32ErrorCodes.ERROR_DS_CANT_ON_RDN:
        Win32ErrorCodeDescription := 'The directory service cannot perform the requested operation on the RDN attribute of an object.';
    Win32ErrorCodes.ERROR_DS_CANT_MOD_OBJ_CLASS:
        Win32ErrorCodeDescription :=
            'The directory service detected an attempt to modify the object class of an object.';
    Win32ErrorCodes.ERROR_DS_CROSS_DOM_MOVE_ERROR:
        Win32ErrorCodeDescription :=
            'The requested cross-domain move operation could not be performed.';
    Win32ErrorCodes.ERROR_DS_GC_NOT_AVAILABLE:
        Win32ErrorCodeDescription := 'Unable to contact the global catalog server.';
    Win32ErrorCodes.ERROR_SHARED_POLICY:
        Win32ErrorCodeDescription :=
            'The policy object is shared and can only be modified at the root.';
    Win32ErrorCodes.ERROR_POLICY_OBJECT_NOT_FOUND:
        Win32ErrorCodeDescription := 'The policy object does not exist.';
    Win32ErrorCodes.ERROR_POLICY_ONLY_IN_DS:
        Win32ErrorCodeDescription :=
            'The requested policy information is only in the directory service.';
    Win32ErrorCodes.ERROR_PROMOTION_ACTIVE:
        Win32ErrorCodeDescription := 'A domain controller promotion is currently active.';
    Win32ErrorCodes.ERROR_NO_PROMOTION_ACTIVE:
        Win32ErrorCodeDescription := 'A domain controller promotion is not currently active';
    Win32ErrorCodes.ERROR_DS_OPERATIONS_ERROR:
        Win32ErrorCodeDescription := 'An operations error occurred.';
    Win32ErrorCodes.ERROR_DS_PROTOCOL_ERROR:
        Win32ErrorCodeDescription := 'A protocol error occurred.';
    Win32ErrorCodes.ERROR_DS_TIMELIMIT_EXCEEDED:
        Win32ErrorCodeDescription := 'The time limit for this request was exceeded.';
    Win32ErrorCodes.ERROR_DS_SIZELIMIT_EXCEEDED:
        Win32ErrorCodeDescription := 'The size limit for this request was exceeded.';
    Win32ErrorCodes.ERROR_DS_ADMIN_LIMIT_EXCEEDED:
        Win32ErrorCodeDescription := 'The administrative limit for this request was exceeded.';
    Win32ErrorCodes.ERROR_DS_COMPARE_FALSE:
        Win32ErrorCodeDescription := 'The compare response was false.';
    Win32ErrorCodes.ERROR_DS_COMPARE_TRUE:
        Win32ErrorCodeDescription := 'The compare response was true.';
    Win32ErrorCodes.ERROR_DS_AUTH_METHOD_NOT_SUPPORTED:
        Win32ErrorCodeDescription :=
            'The requested authentication method is not supported by the server.';
    Win32ErrorCodes.ERROR_DS_STRONG_AUTH_REQUIRED:
        Win32ErrorCodeDescription :=
            'A more secure authentication method is required for this server.';
    Win32ErrorCodes.ERROR_DS_INAPPROPRIATE_AUTH:
        Win32ErrorCodeDescription := 'Inappropriate authentication.';
    Win32ErrorCodes.ERROR_DS_AUTH_UNKNOWN:
        Win32ErrorCodeDescription := 'The authentication mechanism is unknown.';
    Win32ErrorCodes.ERROR_DS_REFERRAL:
        Win32ErrorCodeDescription := 'A referral was returned from the server.';
    Win32ErrorCodes.ERROR_DS_UNAVAILABLE_CRIT_EXTENSION:
        Win32ErrorCodeDescription :=
            'The server does not support the requested critical extension.';
    Win32ErrorCodes.ERROR_DS_CONFIDENTIALITY_REQUIRED:
        Win32ErrorCodeDescription := 'This request requires a secure connection.';
    Win32ErrorCodes.ERROR_DS_INAPPROPRIATE_MATCHING:
        Win32ErrorCodeDescription := 'Inappropriate matching.';
    Win32ErrorCodes.ERROR_DS_CONSTRAINT_VIOLATION:
        Win32ErrorCodeDescription := 'A constraint violation occurred.';
    Win32ErrorCodes.ERROR_DS_NO_SUCH_OBJECT:
        Win32ErrorCodeDescription := 'There is no such object on the server.';
    Win32ErrorCodes.ERROR_DS_ALIAS_PROBLEM:
        Win32ErrorCodeDescription := 'There is an alias problem.';
    Win32ErrorCodes.ERROR_DS_INVALID_DN_SYNTAX:
        Win32ErrorCodeDescription := 'An invalid dn syntax has been specified.';
    Win32ErrorCodes.ERROR_DS_IS_LEAF:
        Win32ErrorCodeDescription := 'The object is a leaf object.';
    Win32ErrorCodes.ERROR_DS_ALIAS_DEREF_PROBLEM:
        Win32ErrorCodeDescription := 'There is an alias dereferencing problem.';
    Win32ErrorCodes.ERROR_DS_UNWILLING_TO_PERFORM:
        Win32ErrorCodeDescription := 'The server is unwilling to process the request.';
    Win32ErrorCodes.ERROR_DS_LOOP_DETECT:
        Win32ErrorCodeDescription := 'A loop has been detected.';
    Win32ErrorCodes.ERROR_DS_NAMING_VIOLATION:
        Win32ErrorCodeDescription := 'There is a naming violation.';
    Win32ErrorCodes.ERROR_DS_OBJECT_RESULTS_TOO_LARGE:
        Win32ErrorCodeDescription := 'The result set is too large.';
    Win32ErrorCodes.ERROR_DS_AFFECTS_MULTIPLE_DSAS:
        Win32ErrorCodeDescription := 'The operation affects multiple DSAs';
    Win32ErrorCodes.ERROR_DS_SERVER_DOWN:
        Win32ErrorCodeDescription := 'The server is not operational.';
    Win32ErrorCodes.ERROR_DS_LOCAL_ERROR:
        Win32ErrorCodeDescription := 'A local error has occurred.';
    Win32ErrorCodes.ERROR_DS_ENCODING_ERROR:
        Win32ErrorCodeDescription := 'An encoding error has occurred.';
    Win32ErrorCodes.ERROR_DS_DECODING_ERROR:
        Win32ErrorCodeDescription := 'A decoding error has occurred.';
    Win32ErrorCodes.ERROR_DS_FILTER_UNKNOWN:
        Win32ErrorCodeDescription := 'The search filter cannot be recognized.';
    Win32ErrorCodes.ERROR_DS_PARAM_ERROR:
        Win32ErrorCodeDescription := 'One or more parameters are illegal.';
    Win32ErrorCodes.ERROR_DS_NOT_SUPPORTED:
        Win32ErrorCodeDescription := 'The specified method is not supported.';
    Win32ErrorCodes.ERROR_DS_NO_RESULTS_RETURNED:
        Win32ErrorCodeDescription := 'No results were returned.';
    Win32ErrorCodes.ERROR_DS_CONTROL_NOT_FOUND:
        Win32ErrorCodeDescription := 'The specified control is not supported by the server.';
    Win32ErrorCodes.ERROR_DS_CLIENT_LOOP:
        Win32ErrorCodeDescription := 'A referral loop was detected by the client.';
    Win32ErrorCodes.ERROR_DS_REFERRAL_LIMIT_EXCEEDED:
        Win32ErrorCodeDescription := 'The preset referral limit was exceeded.';
    Win32ErrorCodes.ERROR_DS_SORT_CONTROL_MISSING:
        Win32ErrorCodeDescription := 'The search requires a SORT control.';
    Win32ErrorCodes.ERROR_DS_OFFSET_RANGE_ERROR:
        Win32ErrorCodeDescription := 'The search results exceed the offset range specified.';
    Win32ErrorCodes.ERROR_DS_ROOT_MUST_BE_NC:
        Win32ErrorCodeDescription := 'The root object must be the head of a naming context. The root object cannot have an instantiated parent.';
    Win32ErrorCodes.ERROR_DS_ADD_REPLICA_INHIBITED:
        Win32ErrorCodeDescription := 'The add replica operation cannot be performed. The naming context must be writable in order to create the replica.';
    Win32ErrorCodes.ERROR_DS_ATT_NOT_DEF_IN_SCHEMA:
        Win32ErrorCodeDescription :=
            'A reference to an attribute that is not defined in the schema occurred.';
    Win32ErrorCodes.ERROR_DS_MAX_OBJ_SIZE_EXCEEDED:
        Win32ErrorCodeDescription := 'The maximum size of an object has been exceeded.';
    Win32ErrorCodes.ERROR_DS_OBJ_STRING_NAME_EXISTS:
        Win32ErrorCodeDescription :=
            'An attempt was made to add an object to the directory with a name that is already in use.';
    Win32ErrorCodes.ERROR_DS_NO_RDN_DEFINED_IN_SCHEMA:
        Win32ErrorCodeDescription := 'An attempt was made to add an object of a class that does not have an RDN defined in the schema.';
    Win32ErrorCodes.ERROR_DS_RDN_DOESNT_MATCH_SCHEMA:
        Win32ErrorCodeDescription := 'An attempt was made to add an object using an RDN that is not the RDN defined in the schema.';
    Win32ErrorCodes.ERROR_DS_NO_REQUESTED_ATTS_FOUND:
        Win32ErrorCodeDescription := 'None of the requested attributes were found on the objects.';
    Win32ErrorCodes.ERROR_DS_USER_BUFFER_TO_SMALL:
        Win32ErrorCodeDescription := 'The user buffer is too small.';
    Win32ErrorCodes.ERROR_DS_ATT_IS_NOT_ON_OBJ:
        Win32ErrorCodeDescription :=
            'The attribute specified in the operation is not present on the object.';
    Win32ErrorCodes.ERROR_DS_ILLEGAL_MOD_OPERATION:
        Win32ErrorCodeDescription :=
            'Illegal modify operation. Some aspect of the modification is not permitted.';
    Win32ErrorCodes.ERROR_DS_OBJ_TOO_LARGE:
        Win32ErrorCodeDescription := 'The specified object is too large.';
    Win32ErrorCodes.ERROR_DS_BAD_INSTANCE_TYPE:
        Win32ErrorCodeDescription := 'The specified instance type is not valid.';
    Win32ErrorCodes.ERROR_DS_MASTERDSA_REQUIRED:
        Win32ErrorCodeDescription := 'The operation must be performed at a master DSA.';
    Win32ErrorCodes.ERROR_DS_OBJECT_CLASS_REQUIRED:
        Win32ErrorCodeDescription := 'The object class attribute must be specified.';
    Win32ErrorCodes.ERROR_DS_MISSING_REQUIRED_ATT:
        Win32ErrorCodeDescription := 'A required attribute is missing.';
    Win32ErrorCodes.ERROR_DS_ATT_NOT_DEF_FOR_CLASS:
        Win32ErrorCodeDescription := 'An attempt was made to modify an object to include an attribute that is not legal for its class';
    Win32ErrorCodes.ERROR_DS_ATT_ALREADY_EXISTS:
        Win32ErrorCodeDescription := 'The specified attribute is already present on the object.';
    Win32ErrorCodes.ERROR_DS_CANT_ADD_ATT_VALUES:
        Win32ErrorCodeDescription := 'The specified attribute is not present, or has no values.';
    Win32ErrorCodes.ERROR_DS_SINGLE_VALUE_CONSTRAINT:
        Win32ErrorCodeDescription :=
            'Multiple values were specified for an attribute that can have only one value.';
    Win32ErrorCodes.ERROR_DS_RANGE_CONSTRAINT:
        Win32ErrorCodeDescription :=
            'A value for the attribute was not in the acceptable range of values.';
    Win32ErrorCodes.ERROR_DS_ATT_VAL_ALREADY_EXISTS:
        Win32ErrorCodeDescription := 'The specified value already exists.';
    Win32ErrorCodes.ERROR_DS_CANT_REM_MISSING_ATT:
        Win32ErrorCodeDescription :=
            'The attribute cannot be removed because it is not present on the object.';
    Win32ErrorCodes.ERROR_DS_CANT_REM_MISSING_ATT_VAL:
        Win32ErrorCodeDescription :=
            'The attribute value cannot be removed because it is not present on the object.';
    Win32ErrorCodes.ERROR_DS_ROOT_CANT_BE_SUBREF:
        Win32ErrorCodeDescription := 'The specified root object cannot be a subref.';
    Win32ErrorCodes.ERROR_DS_NO_CHAINING:
        Win32ErrorCodeDescription := 'Chaining is not permitted.';
    Win32ErrorCodes.ERROR_DS_NO_CHAINED_EVAL:
        Win32ErrorCodeDescription := 'Chained evaluation is not permitted.';
    Win32ErrorCodes.ERROR_DS_NO_PARENT_OBJECT:
        Win32ErrorCodeDescription := 'The operation could not be performed because the objects parent is either uninstantiated or deleted.';
    Win32ErrorCodes.ERROR_DS_PARENT_IS_AN_ALIAS:
        Win32ErrorCodeDescription :=
            'Having a parent that is an alias is not permitted. Aliases are leaf objects.';
    Win32ErrorCodes.ERROR_DS_CANT_MIX_MASTER_AND_REPS:
        Win32ErrorCodeDescription :=
            'The object and parent must be of the same type, either both masters or both replicas.';
    Win32ErrorCodes.ERROR_DS_CHILDREN_EXIST:
        Win32ErrorCodeDescription := 'The operation cannot be performed because child objects exist. This operation can only be performed on a leaf object.';
    Win32ErrorCodes.ERROR_DS_OBJ_NOT_FOUND:
        Win32ErrorCodeDescription := 'Directory object not found.';
    Win32ErrorCodes.ERROR_DS_ALIASED_OBJ_MISSING:
        Win32ErrorCodeDescription := 'The aliased object is missing.';
    Win32ErrorCodes.ERROR_DS_BAD_NAME_SYNTAX:
        Win32ErrorCodeDescription := 'The object name has bad syntax.';
    Win32ErrorCodes.ERROR_DS_ALIAS_POINTS_TO_ALIAS:
        Win32ErrorCodeDescription := 'It is not permitted for an alias to refer to another alias.';
    Win32ErrorCodes.ERROR_DS_CANT_DEREF_ALIAS:
        Win32ErrorCodeDescription := 'The alias cannot be dereferenced.';
    Win32ErrorCodes.ERROR_DS_OUT_OF_SCOPE:
        Win32ErrorCodeDescription := 'The operation is out of scope.';
    Win32ErrorCodes.ERROR_DS_OBJECT_BEING_REMOVED:
        Win32ErrorCodeDescription :=
            'The operation cannot continue because the object is in the process of being removed.';
    Win32ErrorCodes.ERROR_DS_CANT_DELETE_DSA_OBJ:
        Win32ErrorCodeDescription := 'The DSA object cannot be deleted.';
    Win32ErrorCodes.ERROR_DS_GENERIC_ERROR:
        Win32ErrorCodeDescription := 'A directory service error has occurred.';
    Win32ErrorCodes.ERROR_DS_DSA_MUST_BE_INT_MASTER:
        Win32ErrorCodeDescription :=
            'The operation can only be performed on an internal master DSA object.';
    Win32ErrorCodes.ERROR_DS_CLASS_NOT_DSA:
        Win32ErrorCodeDescription := 'The object must be of class DSA.';
    Win32ErrorCodes.ERROR_DS_INSUFF_ACCESS_RIGHTS:
        Win32ErrorCodeDescription := 'Insufficient access rights to perform the operation.';
    Win32ErrorCodes.ERROR_DS_ILLEGAL_SUPERIOR:
        Win32ErrorCodeDescription :=
            'The object cannot be added because the parent is not on the list of possible superiors.';
    Win32ErrorCodes.ERROR_DS_ATTRIBUTE_OWNED_BY_SAM:
        Win32ErrorCodeDescription := 'Access to the attribute is not permitted because the attribute is owned by the Security Accounts Manager (SAM).';
    Win32ErrorCodes.ERROR_DS_NAME_TOO_MANY_PARTS:
        Win32ErrorCodeDescription := 'The name has too many parts.';
    Win32ErrorCodes.ERROR_DS_NAME_TOO_LONG:
        Win32ErrorCodeDescription := 'The name is too long.';
    Win32ErrorCodes.ERROR_DS_NAME_VALUE_TOO_LONG:
        Win32ErrorCodeDescription := 'The name value is too long.';
    Win32ErrorCodes.ERROR_DS_NAME_UNPARSEABLE:
        Win32ErrorCodeDescription := 'The directory service encountered an error parsing a name.';
    Win32ErrorCodes.ERROR_DS_NAME_TYPE_UNKNOWN:
        Win32ErrorCodeDescription :=
            'The directory service cannot get the attribute type for a name.';
    Win32ErrorCodes.ERROR_DS_NOT_AN_OBJECT:
        Win32ErrorCodeDescription :=
            'The name does not identify an object; the name identifies a phantom.';
    Win32ErrorCodes.ERROR_DS_SEC_DESC_TOO_SHORT:
        Win32ErrorCodeDescription := 'The security descriptor is too short.';
    Win32ErrorCodes.ERROR_DS_SEC_DESC_INVALID:
        Win32ErrorCodeDescription := 'The security descriptor is invalid.';
    Win32ErrorCodes.ERROR_DS_NO_DELETED_NAME:
        Win32ErrorCodeDescription := 'Failed to create name for deleted object.';
    Win32ErrorCodes.ERROR_DS_SUBREF_MUST_HAVE_PARENT:
        Win32ErrorCodeDescription := 'The parent of a new subref must exist.';
    Win32ErrorCodes.ERROR_DS_NCNAME_MUST_BE_NC:
        Win32ErrorCodeDescription := 'The object must be a naming context.';
    Win32ErrorCodes.ERROR_DS_CANT_ADD_SYSTEM_ONLY:
        Win32ErrorCodeDescription :=
            'It is not permitted to add an attribute which is owned by the system.';
    Win32ErrorCodes.ERROR_DS_CLASS_MUST_BE_CONCRETE:
        Win32ErrorCodeDescription :=
            'The class of the object must be structural; you cannot instantiate an abstract class.';
    Win32ErrorCodes.ERROR_DS_INVALID_DMD:
        Win32ErrorCodeDescription := 'The schema object could not be found.';
    Win32ErrorCodes.ERROR_DS_OBJ_GUID_EXISTS:
        Win32ErrorCodeDescription :=
            'A local object with this GUID (dead or alive) already exists.';
    Win32ErrorCodes.ERROR_DS_NOT_ON_BACKLINK:
        Win32ErrorCodeDescription := 'The operation cannot be performed on a back link.';
    Win32ErrorCodes.ERROR_DS_NO_CROSSREF_FOR_NC:
        Win32ErrorCodeDescription :=
            'The cross reference for the specified naming context could not be found.';
    Win32ErrorCodes.ERROR_DS_SHUTTING_DOWN:
        Win32ErrorCodeDescription :=
            'The operation could not be performed because the directory service is shutting down.';
    Win32ErrorCodes.ERROR_DS_UNKNOWN_OPERATION:
        Win32ErrorCodeDescription := 'The directory service request is invalid.';
    Win32ErrorCodes.ERROR_DS_INVALID_ROLE_OWNER:
        Win32ErrorCodeDescription := 'The role owner attribute could not be read.';
    Win32ErrorCodes.ERROR_DS_COULDNT_CONTACT_FSMO:
        Win32ErrorCodeDescription :=
            'The requested FSMO operation failed. The current FSMO holder could not be reached.';
    Win32ErrorCodes.ERROR_DS_CROSS_NC_DN_RENAME:
        Win32ErrorCodeDescription :=
            'Modification of a DN across a naming context is not permitted.';
    Win32ErrorCodes.ERROR_DS_CANT_MOD_SYSTEM_ONLY:
        Win32ErrorCodeDescription :=
            'The attribute cannot be modified because it is owned by the system.';
    Win32ErrorCodes.ERROR_DS_REPLICATOR_ONLY:
        Win32ErrorCodeDescription := 'Only the replicator can perform this function.';
    Win32ErrorCodes.ERROR_DS_OBJ_CLASS_NOT_DEFINED:
        Win32ErrorCodeDescription := 'The specified class is not defined.';
    Win32ErrorCodes.ERROR_DS_OBJ_CLASS_NOT_SUBCLASS:
        Win32ErrorCodeDescription := 'The specified class is not a subclass.';
    Win32ErrorCodes.ERROR_DS_NAME_REFERENCE_INVALID:
        Win32ErrorCodeDescription := 'The name reference is invalid.';
    Win32ErrorCodes.ERROR_DS_CROSS_REF_EXISTS:
        Win32ErrorCodeDescription := 'A cross reference already exists.';
    Win32ErrorCodes.ERROR_DS_CANT_DEL_MASTER_CROSSREF:
        Win32ErrorCodeDescription := 'It is not permitted to delete a master cross reference.';
    Win32ErrorCodes.ERROR_DS_SUBTREE_NOTIFY_NOT_NC_HEAD:
        Win32ErrorCodeDescription := 'Subtree notifications are only supported on NC heads.';
    Win32ErrorCodes.ERROR_DS_NOTIFY_FILTER_TOO_COMPLEX:
        Win32ErrorCodeDescription := 'Notification filter is too complex.';
    Win32ErrorCodes.ERROR_DS_DUP_RDN:
        Win32ErrorCodeDescription := 'Schema update failed: duplicate RDN.';
    Win32ErrorCodes.ERROR_DS_DUP_OID:
        Win32ErrorCodeDescription := 'Schema update failed: duplicate OID';
    Win32ErrorCodes.ERROR_DS_DUP_MAPI_ID:
        Win32ErrorCodeDescription := 'Schema update failed: duplicate MAPI identifier.';
    Win32ErrorCodes.ERROR_DS_DUP_SCHEMA_ID_GUID:
        Win32ErrorCodeDescription := 'Schema update failed: duplicate schema-id GUID.';
    Win32ErrorCodes.ERROR_DS_DUP_LDAP_DISPLAY_NAME:
        Win32ErrorCodeDescription := 'Schema update failed: duplicate LDAP display name.';
    Win32ErrorCodes.ERROR_DS_SEMANTIC_ATT_TEST:
        Win32ErrorCodeDescription := 'Schema update failed: range-lower less than range upper';
    Win32ErrorCodes.ERROR_DS_SYNTAX_MISMATCH:
        Win32ErrorCodeDescription := 'Schema update failed: syntax mismatch';
    Win32ErrorCodes.ERROR_DS_EXISTS_IN_MUST_HAVE:
        Win32ErrorCodeDescription := 'Schema deletion failed: attribute is used in must-contain';
    Win32ErrorCodes.ERROR_DS_EXISTS_IN_MAY_HAVE:
        Win32ErrorCodeDescription := 'Schema deletion failed: attribute is used in may-contain';
    Win32ErrorCodes.ERROR_DS_NONEXISTENT_MAY_HAVE:
        Win32ErrorCodeDescription :=
            'Schema update failed: attribute in may-contain does not exist';
    Win32ErrorCodes.ERROR_DS_NONEXISTENT_MUST_HAVE:
        Win32ErrorCodeDescription :=
            'Schema update failed: attribute in must-contain does not exist';
    Win32ErrorCodes.ERROR_DS_AUX_CLS_TEST_FAIL:
        Win32ErrorCodeDescription :=
            'Schema update failed: class in aux-class list does not exist or is not an auxiliary class';
    Win32ErrorCodes.ERROR_DS_NONEXISTENT_POSS_SUP:
        Win32ErrorCodeDescription :=
            'Schema update failed: class in poss-superiors does not exist';
    Win32ErrorCodes.ERROR_DS_SUB_CLS_TEST_FAIL:
        Win32ErrorCodeDescription := 'Schema update failed: class in subclassof list does not exist or does not satisfy hierarchy rules';
    Win32ErrorCodes.ERROR_DS_BAD_RDN_ATT_ID_SYNTAX:
        Win32ErrorCodeDescription := 'Schema update failed: Rdn-Att-Id has wrong syntax';
    Win32ErrorCodes.ERROR_DS_EXISTS_IN_AUX_CLS:
        Win32ErrorCodeDescription := 'Schema deletion failed: class is used as auxiliary class';
    Win32ErrorCodes.ERROR_DS_EXISTS_IN_SUB_CLS:
        Win32ErrorCodeDescription := 'Schema deletion failed: class is used as sub class';
    Win32ErrorCodes.ERROR_DS_EXISTS_IN_POSS_SUP:
        Win32ErrorCodeDescription := 'Schema deletion failed: class is used as poss superior';
    Win32ErrorCodes.ERROR_DS_RECALCSCHEMA_FAILED:
        Win32ErrorCodeDescription := 'Schema update failed in recalculating validation cache.';
    Win32ErrorCodes.ERROR_DS_TREE_DELETE_NOT_FINISHED:
        Win32ErrorCodeDescription := 'The tree deletion is not finished.';
    Win32ErrorCodes.ERROR_DS_CANT_DELETE:
        Win32ErrorCodeDescription := 'The requested delete operation could not be performed.';
    Win32ErrorCodes.ERROR_DS_ATT_SCHEMA_REQ_ID:
        Win32ErrorCodeDescription :=
            'Cannot read the governs class identifier for the schema record.';
    Win32ErrorCodes.ERROR_DS_BAD_ATT_SCHEMA_SYNTAX:
        Win32ErrorCodeDescription := 'The attribute schema has bad syntax.';
    Win32ErrorCodes.ERROR_DS_CANT_CACHE_ATT:
        Win32ErrorCodeDescription := 'The attribute could not be cached.';
    Win32ErrorCodes.ERROR_DS_CANT_CACHE_CLASS:
        Win32ErrorCodeDescription := 'The class could not be cached.';
    Win32ErrorCodes.ERROR_DS_CANT_REMOVE_ATT_CACHE:
        Win32ErrorCodeDescription := 'The attribute could not be removed from the cache.';
    Win32ErrorCodes.ERROR_DS_CANT_REMOVE_CLASS_CACHE:
        Win32ErrorCodeDescription := 'The class could not be removed from the cache.';
    Win32ErrorCodes.ERROR_DS_CANT_RETRIEVE_DN:
        Win32ErrorCodeDescription := 'The distinguished name attribute could not be read.';
    Win32ErrorCodes.ERROR_DS_MISSING_SUPREF:
        Win32ErrorCodeDescription := 'A required subref is missing.';
    Win32ErrorCodes.ERROR_DS_CANT_RETRIEVE_INSTANCE:
        Win32ErrorCodeDescription := 'The instance type attribute could not be retrieved.';
    Win32ErrorCodes.ERROR_DS_CODE_INCONSISTENCY:
        Win32ErrorCodeDescription := 'An internal error has occurred.';
    Win32ErrorCodes.ERROR_DS_DATABASE_ERROR:
        Win32ErrorCodeDescription := 'A database error has occurred.';
    Win32ErrorCodes.ERROR_DS_GOVERNSID_MISSING:
        Win32ErrorCodeDescription := 'The attribute GOVERNSID is missing.';
    Win32ErrorCodes.ERROR_DS_MISSING_EXPECTED_ATT:
        Win32ErrorCodeDescription := 'An expected attribute is missing.';
    Win32ErrorCodes.ERROR_DS_NCNAME_MISSING_CR_REF:
        Win32ErrorCodeDescription := 'The specified naming context is missing a cross reference.';
    Win32ErrorCodes.ERROR_DS_SECURITY_CHECKING_ERROR:
        Win32ErrorCodeDescription := 'A security checking error has occurred.';
    Win32ErrorCodes.ERROR_DS_SCHEMA_NOT_LOADED:
        Win32ErrorCodeDescription := 'The schema is not loaded.';
    Win32ErrorCodes.ERROR_DS_SCHEMA_ALLOC_FAILED:
        Win32ErrorCodeDescription :=
            'Schema allocation failed. Please check if the machine is running low on memory.';
    Win32ErrorCodes.ERROR_DS_ATT_SCHEMA_REQ_SYNTAX:
        Win32ErrorCodeDescription :=
            'Failed to obtain the required syntax for the attribute schema.';
    Win32ErrorCodes.ERROR_DS_GCVERIFY_ERROR:
        Win32ErrorCodeDescription := 'The global catalog verification failed. The global catalog is not available or does not support the operation. Some part of the directory is currently not available.';
    Win32ErrorCodes.ERROR_DS_DRA_SCHEMA_MISMATCH:
        Win32ErrorCodeDescription := 'The replication operation failed because of a schema mismatch between the servers involved.';
    Win32ErrorCodes.ERROR_DS_CANT_FIND_DSA_OBJ:
        Win32ErrorCodeDescription := 'The DSA object could not be found.';
    Win32ErrorCodes.ERROR_DS_CANT_FIND_EXPECTED_NC:
        Win32ErrorCodeDescription := 'The naming context could not be found.';
    Win32ErrorCodes.ERROR_DS_CANT_FIND_NC_IN_CACHE:
        Win32ErrorCodeDescription := 'The naming context could not be found in the cache.';
    Win32ErrorCodes.ERROR_DS_CANT_RETRIEVE_CHILD:
        Win32ErrorCodeDescription := 'The child object could not be retrieved.';
    Win32ErrorCodes.ERROR_DS_SECURITY_ILLEGAL_MODIFY:
        Win32ErrorCodeDescription := 'The modification was not permitted for security reasons.';
    Win32ErrorCodes.ERROR_DS_CANT_REPLACE_HIDDEN_REC:
        Win32ErrorCodeDescription := 'The operation cannot replace the hidden record.';
    Win32ErrorCodes.ERROR_DS_BAD_HIERARCHY_FILE:
        Win32ErrorCodeDescription := 'The hierarchy file is invalid.';
    Win32ErrorCodes.ERROR_DS_BUILD_HIERARCHY_TABLE_FAILED:
        Win32ErrorCodeDescription := 'The attempt to build the hierarchy table failed.';
    Win32ErrorCodes.ERROR_DS_CONFIG_PARAM_MISSING:
        Win32ErrorCodeDescription :=
            'The directory configuration parameter is missing from the registry.';
    Win32ErrorCodes.ERROR_DS_COUNTING_AB_INDICES_FAILED:
        Win32ErrorCodeDescription := 'The attempt to count the address book indices failed.';
    Win32ErrorCodes.ERROR_DS_HIERARCHY_TABLE_MALLOC_FAILED:
        Win32ErrorCodeDescription := 'The allocation of the hierarchy table failed.';
    Win32ErrorCodes.ERROR_DS_INTERNAL_FAILURE:
        Win32ErrorCodeDescription := 'The directory service encountered an internal failure.';
    Win32ErrorCodes.ERROR_DS_UNKNOWN_ERROR:
        Win32ErrorCodeDescription := 'The directory service encountered an unknown failure.';
    Win32ErrorCodes.ERROR_DS_ROOT_REQUIRES_CLASS_TOP:
        Win32ErrorCodeDescription := 'A root object requires a class of top.';
    Win32ErrorCodes.ERROR_DS_REFUSING_FSMO_ROLES:
        Win32ErrorCodeDescription := 'This directory server is shutting down, and cannot take ownership of new floating single-master operation roles.';
    Win32ErrorCodes.ERROR_DS_MISSING_FSMO_SETTINGS:
        Win32ErrorCodeDescription := 'The directory service is missing mandatory configuration information, and is unable to determine the ownership of floating single-master operation roles.';
    Win32ErrorCodes.ERROR_DS_UNABLE_TO_SURRENDER_ROLES:
        Win32ErrorCodeDescription := 'The directory service was unable to transfer ownership of one or more floating single-master operation roles to other servers.';
    Win32ErrorCodes.ERROR_DS_DRA_GENERIC:
        Win32ErrorCodeDescription := 'The replication operation failed.';
    Win32ErrorCodes.ERROR_DS_DRA_INVALID_PARAMETER:
        Win32ErrorCodeDescription :=
            'An invalid parameter was specified for this replication operation.';
    Win32ErrorCodes.ERROR_DS_DRA_BUSY:
        Win32ErrorCodeDescription :=
            'The directory service is too busy to complete the replication operation at this time.';
    Win32ErrorCodes.ERROR_DS_DRA_BAD_DN:
        Win32ErrorCodeDescription :=
            'The distinguished name specified for this replication operation is invalid.';
    Win32ErrorCodes.ERROR_DS_DRA_BAD_NC:
        Win32ErrorCodeDescription :=
            'The naming context specified for this replication operation is invalid.';
    Win32ErrorCodes.ERROR_DS_DRA_DN_EXISTS:
        Win32ErrorCodeDescription :=
            'The distinguished name specified for this replication operation already exists.';
    Win32ErrorCodes.ERROR_DS_DRA_INTERNAL_ERROR:
        Win32ErrorCodeDescription := 'The replication system encountered an internal error.';
    Win32ErrorCodes.ERROR_DS_DRA_INCONSISTENT_DIT:
        Win32ErrorCodeDescription :=
            'The replication operation encountered a database inconsistency.';
    Win32ErrorCodes.ERROR_DS_DRA_CONNECTION_FAILED:
        Win32ErrorCodeDescription :=
            'The server specified for this replication operation could not be contacted.';
    Win32ErrorCodes.ERROR_DS_DRA_BAD_INSTANCE_TYPE:
        Win32ErrorCodeDescription :=
            'The replication operation encountered an object with an invalid instance type.';
    Win32ErrorCodes.ERROR_DS_DRA_OUT_OF_MEM:
        Win32ErrorCodeDescription := 'The replication operation failed to allocate memory.';
    Win32ErrorCodes.ERROR_DS_DRA_MAIL_PROBLEM:
        Win32ErrorCodeDescription :=
            'The replication operation encountered an error with the mail system.';
    Win32ErrorCodes.ERROR_DS_DRA_REF_ALREADY_EXISTS:
        Win32ErrorCodeDescription :=
            'The replication reference information for the target server already exists.';
    Win32ErrorCodes.ERROR_DS_DRA_REF_NOT_FOUND:
        Win32ErrorCodeDescription :=
            'The replication reference information for the target server does not exist.';
    Win32ErrorCodes.ERROR_DS_DRA_OBJ_IS_REP_SOURCE:
        Win32ErrorCodeDescription :=
            'The naming context cannot be removed because it is replicated to another server.';
    Win32ErrorCodes.ERROR_DS_DRA_DB_ERROR:
        Win32ErrorCodeDescription := 'The replication operation encountered a database error.';
    Win32ErrorCodes.ERROR_DS_DRA_NO_REPLICA:
        Win32ErrorCodeDescription := 'The naming context is in the process of being removed or is not replicated from the specified server.';
    Win32ErrorCodes.ERROR_DS_DRA_ACCESS_DENIED:
        Win32ErrorCodeDescription := 'Replication access was denied.';
    Win32ErrorCodes.ERROR_DS_DRA_NOT_SUPPORTED:
        Win32ErrorCodeDescription :=
            'The requested operation is not supported by this version of the directory service.';
    Win32ErrorCodes.ERROR_DS_DRA_RPC_CANCELLED:
        Win32ErrorCodeDescription := 'The replication remote procedure call was cancelled.';
    Win32ErrorCodes.ERROR_DS_DRA_SOURCE_DISABLED:
        Win32ErrorCodeDescription :=
            'The source server is currently rejecting replication requests.';
    Win32ErrorCodes.ERROR_DS_DRA_SINK_DISABLED:
        Win32ErrorCodeDescription :=
            'The destination server is currently rejecting replication requests.';
    Win32ErrorCodes.ERROR_DS_DRA_NAME_COLLISION:
        Win32ErrorCodeDescription :=
            'The replication operation failed due to a collision of object names.';
    Win32ErrorCodes.ERROR_DS_DRA_SOURCE_REINSTALLED:
        Win32ErrorCodeDescription := 'The replication source has been reinstalled.';
    Win32ErrorCodes.ERROR_DS_DRA_MISSING_PARENT:
        Win32ErrorCodeDescription :=
            'The replication operation failed because a required parent object is missing.';
    Win32ErrorCodes.ERROR_DS_DRA_PREEMPTED:
        Win32ErrorCodeDescription := 'The replication operation was preempted.';
    Win32ErrorCodes.ERROR_DS_DRA_ABANDON_SYNC:
        Win32ErrorCodeDescription :=
            'The replication synchronization attempt was abandoned because of a lack of updates.';
    Win32ErrorCodes.ERROR_DS_DRA_SHUTDOWN:
        Win32ErrorCodeDescription :=
            'The replication operation was terminated because the system is shutting down.';
    Win32ErrorCodes.ERROR_DS_DRA_INCOMPATIBLE_PARTIAL_SET:
        Win32ErrorCodeDescription := 'The replication synchronization attempt failed as the destination partial attribute set is not a subset of source partial attribute set.';
    Win32ErrorCodes.ERROR_DS_DRA_SOURCE_IS_PARTIAL_REPLICA:
        Win32ErrorCodeDescription := 'The replication synchronization attempt failed because a master replica attempted to sync from a partial replica.';
    Win32ErrorCodes.ERROR_DS_DRA_EXTN_CONNECTION_FAILED:
        Win32ErrorCodeDescription := 'The server specified for this replication operation was contacted, but that server was unable to contact an additional server needed to complete the operation.';
    Win32ErrorCodes.ERROR_DS_INSTALL_SCHEMA_MISMATCH:
        Win32ErrorCodeDescription := 'The version of the Active Directory (AD) schema of the source forest is not compatible with the version of AD on this computer. Upgrade the operating system on a domain controller in the source forest before it can be added as a controller to that forest.';
    Win32ErrorCodes.ERROR_DS_DUP_LINK_ID:
        Win32ErrorCodeDescription :=
            'Schema update failed: An attribute with the same link identifier already exists.';
    Win32ErrorCodes.ERROR_DS_NAME_ERROR_RESOLVING:
        Win32ErrorCodeDescription := 'Name translation: Generic processing error.';
    Win32ErrorCodes.ERROR_DS_NAME_ERROR_NOT_FOUND:
        Win32ErrorCodeDescription :=
            'Name translation: Could not find the name or insufficient right to see name.';
    Win32ErrorCodes.ERROR_DS_NAME_ERROR_NOT_UNIQUE:
        Win32ErrorCodeDescription :=
            'Name translation: Input name mapped to more than one output name.';
    Win32ErrorCodes.ERROR_DS_NAME_ERROR_NO_MAPPING:
        Win32ErrorCodeDescription :=
            'Name translation: Input name found, but not the associated output format.';
    Win32ErrorCodes.ERROR_DS_NAME_ERROR_DOMAIN_ONLY:
        Win32ErrorCodeDescription :=
            'Name translation: Unable to resolve completely, only the domain was found.';
    Win32ErrorCodes.ERROR_DS_NAME_ERROR_NO_SYNTACTICAL_MAPPING:
        Win32ErrorCodeDescription := 'Name translation: Unable to perform purely syntactical mapping at the client without going out to the wire.';
    Win32ErrorCodes.ERROR_DS_CONSTRUCTED_ATT_MOD:
        Win32ErrorCodeDescription := 'Modification of a constructed att is not allowed.';
    Win32ErrorCodes.ERROR_DS_WRONG_OM_OBJ_CLASS:
        Win32ErrorCodeDescription :=
            'The OM-Object-Class specified is incorrect for an attribute with the specified syntax.';
    Win32ErrorCodes.ERROR_DS_DRA_REPL_PENDING:
        Win32ErrorCodeDescription := 'The replication request has been posted; waiting for reply.';
    Win32ErrorCodes.ERROR_DS_DS_REQUIRED:
        Win32ErrorCodeDescription :=
            'The requested operation requires a directory service, and none was available.';
    Win32ErrorCodes.ERROR_DS_INVALID_LDAP_DISPLAY_NAME:
        Win32ErrorCodeDescription :=
            'The LDAP display name of the class or attribute contains non-ASCII characters.';
    Win32ErrorCodes.ERROR_DS_NON_BASE_SEARCH:
        Win32ErrorCodeDescription :=
            'The requested search operation is only supported for base searches.';
    Win32ErrorCodes.ERROR_DS_CANT_RETRIEVE_ATTS:
        Win32ErrorCodeDescription := 'The search failed to retrieve attributes from the database.';
    Win32ErrorCodes.ERROR_DS_BACKLINK_WITHOUT_LINK:
        Win32ErrorCodeDescription := 'The schema update operation tried to add a backward link attribute that has no corresponding forward link.';
    Win32ErrorCodes.ERROR_DS_EPOCH_MISMATCH:
        Win32ErrorCodeDescription := 'Source and destination of a cross domain move do not agree on the objects epoch number. Either source or destination does not have the latest version of the object.';
    Win32ErrorCodes.ERROR_DS_SRC_NAME_MISMATCH:
        Win32ErrorCodeDescription := 'Source and destination of a cross domain move do not agree on the objects current name. Either source or destination does not have the latest version of the object.';
    Win32ErrorCodes.ERROR_DS_SRC_AND_DST_NC_IDENTICAL:
        Win32ErrorCodeDescription := 'Source and destination of a cross domain move operation are identical. Caller should use local move operation instead of cross domain move operation.';
    Win32ErrorCodes.ERROR_DS_DST_NC_MISMATCH:
        Win32ErrorCodeDescription := 'Source and destination for a cross domain move are not in agreement on the naming contexts in the forest. Either source or destination does not have the latest version of the Partitions container.';
    Win32ErrorCodes.ERROR_DS_NOT_AUTHORITIVE_FOR_DST_NC:
        Win32ErrorCodeDescription := 'Destination of a cross domain move is not authoritative for the destination naming context.';
    Win32ErrorCodes.ERROR_DS_SRC_GUID_MISMATCH:
        Win32ErrorCodeDescription := 'Source and destination of a cross domain move do not agree on the identity of the source object. Either source or destination does not have the latest version of the source object.';
    Win32ErrorCodes.ERROR_DS_CANT_MOVE_DELETED_OBJECT:
        Win32ErrorCodeDescription := 'Object being moved across domains is already known to be deleted by the destination server. The source server does not have the latest version of the source object.';
    Win32ErrorCodes.ERROR_DS_PDC_OPERATION_IN_PROGRESS:
        Win32ErrorCodeDescription :=
            'Another operation which requires exclusive access to the PDC PSMO is already in progress.';
    Win32ErrorCodes.ERROR_DS_CROSS_DOMAIN_CLEANUP_REQD:
        Win32ErrorCodeDescription := 'A cross domain move operation failed such that the two versions of the moved object exist - one each in the source and destination domains. The destination object needs to be removed to restore the system to a consistent state.';
    Win32ErrorCodes.ERROR_DS_ILLEGAL_XDOM_MOVE_OPERATION:
        Win32ErrorCodeDescription := 'This object may not be moved across domain boundaries either because cross domain moves for this class are disallowed, or the object has some special characteristics, eg: trust account or restricted RID, which prevent its move.';
    Win32ErrorCodes.ERROR_DS_CANT_WITH_ACCT_GROUP_MEMBERSHPS:
        Win32ErrorCodeDescription := 'Cant move objects with memberships across domain boundaries as once moved, this would violate the membership conditions of the account group. Remove the object from any account group memberships and retry.';
    Win32ErrorCodes.ERROR_DS_NC_MUST_HAVE_NC_PARENT:
        Win32ErrorCodeDescription := 'A naming context head must be the immediate child of another naming context head, not of an interior node.';
    Win32ErrorCodes.ERROR_DS_CR_IMPOSSIBLE_TO_VALIDATE:
        Win32ErrorCodeDescription := 'The directory cant validate the proposed naming context name because it doesnt hold a replica of the naming context above the proposed naming context.';
    Win32ErrorCodes.ERROR_DS_DST_DOMAIN_NOT_NATIVE:
        Win32ErrorCodeDescription := 'Destination domain must be in native mode.';
    Win32ErrorCodes.ERROR_DS_MISSING_INFRASTRUCTURE_CONTAINER:
        Win32ErrorCodeDescription := 'The operation can not be performed because the server does not have an infrastructure container in the domain of interest.';
    Win32ErrorCodes.ERROR_DS_CANT_MOVE_ACCOUNT_GROUP:
        Win32ErrorCodeDescription :=
            'Cross-domain move of non-empty account groups is not allowed.';
    Win32ErrorCodes.ERROR_DS_CANT_MOVE_RESOURCE_GROUP:
        Win32ErrorCodeDescription :=
            'Cross-domain move of non-empty resource groups is not allowed.';
    Win32ErrorCodes.ERROR_DS_INVALID_SEARCH_FLAG:
        Win32ErrorCodeDescription := 'The search flags for the attribute are invalid. The ANR bit is valid only on attributes of Unicode or Teletex strings.';
    Win32ErrorCodes.ERROR_DS_NO_TREE_DELETE_ABOVE_NC:
        Win32ErrorCodeDescription := 'Tree deletions starting at an object which has an NC head as a descendant are not allowed.';
    Win32ErrorCodes.ERROR_DS_COULDNT_LOCK_TREE_FOR_DELETE:
        Win32ErrorCodeDescription := 'The directory service failed to lock a tree in preparation for a tree deletion because the tree was in use.';
    Win32ErrorCodes.ERROR_DS_COULDNT_IDENTIFY_OBJECTS_FOR_TREE_DELETE:
        Win32ErrorCodeDescription := 'The directory service failed to identify the list of objects to delete while attempting a tree deletion.';
    Win32ErrorCodes.ERROR_DS_SAM_INIT_FAILURE:
        Win32ErrorCodeDescription := 'Security Accounts Manager initialization failed because of the following error: %1. Error Status: 0x%2. Click OK to shut down the system and reboot into Directory Services Restore Mode. Check the event log for detailed information.';
    Win32ErrorCodes.ERROR_DS_SENSITIVE_GROUP_VIOLATION:
        Win32ErrorCodeDescription :=
            'Only an administrator can modify the membership list of an administrative group.';
    Win32ErrorCodes.ERROR_DS_CANT_MOD_PRIMARYGROUPID:
        Win32ErrorCodeDescription :=
            'Cannot change the primary group ID of a domain controller account.';
    Win32ErrorCodes.ERROR_DS_ILLEGAL_BASE_SCHEMA_MOD:
        Win32ErrorCodeDescription := 'An attempt is made to modify the base schema.';
    Win32ErrorCodes.ERROR_DS_NONSAFE_SCHEMA_CHANGE:
        Win32ErrorCodeDescription := 'Adding a new mandatory attribute to an existing class, deleting one from an existing class, or adding an optional attribute to the special class Top that is not a backlink attribute (directly or through inheritance) is not allowed.';
    Win32ErrorCodes.ERROR_DS_SCHEMA_UPDATE_DISALLOWED:
        Win32ErrorCodeDescription :=
            'Schema update is not allowed on this DC because the DC is not the schema FSMO Role Owner.';
    Win32ErrorCodes.ERROR_DS_CANT_CREATE_UNDER_SCHEMA:
        Win32ErrorCodeDescription := 'An object of this class cannot be created under the schema container. You can only create attribute-schema and class-schema objects under the schema container.';
    Win32ErrorCodes.ERROR_DS_INSTALL_NO_SRC_SCH_VERSION:
        Win32ErrorCodeDescription := 'The replica/child install failed to get the objectVersion attribute on the schema container on the source DC. Either the attribute is missing on the schema container or the credentials supplied do not have permission to read it.';
    Win32ErrorCodes.ERROR_DS_INSTALL_NO_SCH_VERSION_IN_INIFILE:
        Win32ErrorCodeDescription := 'The replica/child install failed to read the objectVersion attribute in the SCHEMA section of the file schema.ini in the system32 directory.';
    Win32ErrorCodes.ERROR_DS_INVALID_GROUP_TYPE:
        Win32ErrorCodeDescription := 'The specified group type is invalid.';
    Win32ErrorCodes.ERROR_DS_NO_NEST_GLOBALGROUP_IN_MIXEDDOMAIN:
        Win32ErrorCodeDescription :=
            'Cannot nest global groups in a mixed domain if the group is security-enabled.';
    Win32ErrorCodes.ERROR_DS_NO_NEST_LOCALGROUP_IN_MIXEDDOMAIN:
        Win32ErrorCodeDescription :=
            'Cannot nest local groups in a mixed domain if the group is security-enabled.';
